# B&R Automation Studio project NAINV104C00R8L515F00 (part 24)

#### Act_Main.st - Do Not Change!!!
```iecst
(** 2020-05-26 **)
ACTION Act_Main:

	//Main
IF bModuleNotOK = FALSE THEN

		CASE eStat OF

			AWActIdle:
				IF eStatus <> Idle THEN	//Reset Data
					//Private
					fbStop(bEn := FALSE);
					fbRstAxisErr(bEn := FALSE);
					fbJog(bEn := FALSE);
					fbMovRel(bEn := FALSE);
					fbMovAbs(bEn := FALSE);
					fbHoming(bEn := FALSE);
					fbPwrOff(bEn := FALSE);
					fbPwrOn(bEn := FALSE);
					fbFullHm(bEn := FALSE);
					fbFullMovAbs(bEn := FALSE);
					fbFullMovAbsBl(bEn := FALSE);
					fbSDOWrite(bEn := FALSE);
					fbTm(IN := FALSE);
					usiStep				:= 0;
					usiCount			:= 0;
					bNotInterruptible	:= FALSE;
					tyParamOutDriver.uiCtrlword_6040.7	:= FALSE;
					sStatTxt	:= a_sStatText[eStat];

				END_IF

				eStatus	:= Idle;

				IF EDGENEG(p_bManual) THEN
					fMotionCANRstCtrlWord(ADR(tyParamOutDriver));
				END_IF

			AWActGoWidth:
				IF (eStatus = Idle OR eStatus = Busy) THEN

					eStatus	:= Busy;

					sStatTxt	:= a_sStatText[eStat];

					bNotInterruptible	:= TRUE;

					CASE usiStep OF
						0:	//Wait For Motion Parameter Update
							p_diMovePosInUM	:= fAWWidthToPosInUM(p_diGoWidth , p_diWidthAtHmPos);
							usiStep	:= 1;

						1:	//Check Position Difference
							IF tyParamOut.bPosDiff = TRUE THEN
								usiStep	:= 2;
							ELSE
								eStatus	:= Done;
							END_IF

						2:	//Move
							fbFullMovAbsBl.tyParamInDriver					:= tyParamInDriver;
							fbFullMovAbsBl.tyParamInMove.diPosInUM			:= p_diMovePosInUM;
							fbFullMovAbsBl.tyParamInMove.diDistInUM			:= p_diMoveDistInUM;
							fbFullMovAbsBl.tyParamInMove.diVelInUMPS		:= p_diMoveVelInUMPS;
							fbFullMovAbsBl.tyParamInMove.diAcc				:= p_diMoveAcc;
							fbFullMovAbsBl.tyParamInMove.diDec				:= p_diMoveDec;
							fbFullMovAbsBl.tyParamOut						:= tyParamOut;
							fbFullMovAbsBl(bEn := TRUE);

							IF fbFullMovAbsBl.udiStatus = 0 THEN
								eStatus	:= Done;
							ELSIF fbFullMovAbsBl.udiStatus < 65534 THEN
								eStatus		:= Error;

								IF fbFullMovAbsBl.udiStatus = 1401 THEN
									udiStatus	:= 10002;	//Power On Time Out While Going New Width
								ELSIF fbFullMovAbsBl.udiStatus = 1402 THEN
									udiStatus	:= 10003;	//Homing Time Out While Going New Width
								ELSIF fbFullMovAbsBl.udiStatus = 1403 THEN
									udiStatus	:= 10004;	//Move Absolute Time Out While Going New Width
								ELSIF fbFullMovAbsBl.udiStatus = 1405 THEN
									udiStatus	:= 10005;	//Stop Motion Time Out While Going New Width
								ELSIF fbFullMovAbsBl.udiStatus = 1408 THEN
									udiStatus	:= 10006;	//Axis Error Reset Failed While Going New Width
								ELSIF fbFullMovAbsBl.udiStatus = 1409 THEN
									udiStatus	:= 10007;	//Axis Error Occur In Move Absolute While Going New Width
								ELSIF fbFullMovAbsBl.udiStatus = 1411 THEN
									udiStatus	:= 10008;	//Axis Error Occur In Homing While Going New Width
								ELSIF fbFullMovAbsBl.udiStatus = 1412 THEN
									udiStatus	:= 10009;	//Homing Done But Home Flag Is Not Activated While Going New Width
								ELSIF fbFullMovAbsBl.udiStatus = 1413 THEN
									udiStatus	:= 10010;	//Forward Limit Activated In Homing While Going New Width
								ELSIF fbFullMovAbsBl.udiStatus = 1414 THEN
									udiStatus	:= 10011;	//Reverse Limit Activated In Homing While Going New Width
								ELSIF fbFullMovAbsBl.udiStatus = 1415 THEN
									udiStatus	:= 10012;	//Forward Limit Activated In Move Absolute While Going New Width
								ELSIF fbFullMovAbsBl.udiStatus = 1416 THEN
									udiStatus	:= 10013;	//Reverse Limit Activated In Move Absolute While Going New Width
								ELSE
									udiStatus	:= fbFullMovAbsBl.udiStatus;
								END_IF
							END_IF

					END_CASE

				END_IF

			AWActGoWidthOff:
				IF (eStatus = Idle OR eStatus = Busy) THEN

					eStatus	:= Busy;

					sStatTxt	:= a_sStatText[eStat];

					bNotInterruptible	:= TRUE;

					CASE usiStep OF
						0:	//Wait For Motion Parameter Update
							p_diMovePosInUM	:= fAWWidthToPosInUM(p_diGoWidth , p_diWidthAtHmPos);
							usiStep	:= 1;

						1:	//Check Position Difference
							IF tyParamOut.bPosDiff = TRUE THEN
								usiStep	:= 2;
							ELSE
								eStatus	:= Done;
							END_IF

						2:	//Move
							fbFullMovAbsBl.tyParamInDriver					:= tyParamInDriver;
							fbFullMovAbsBl.tyParamInMove.diPosInUM			:= p_diMovePosInUM;
							fbFullMovAbsBl.tyParamInMove.diDistInUM			:= p_diMoveDistInUM;
							fbFullMovAbsBl.tyParamInMove.diVelInUMPS		:= p_diMoveVelInUMPS;
							fbFullMovAbsBl.tyParamInMove.diAcc				:= p_diMoveAcc;
							fbFullMovAbsBl.tyParamInMove.diDec				:= p_diMoveDec;
							fbFullMovAbsBl.tyParamOut						:= tyParamOut;
							fbFullMovAbsBl(bEn := TRUE);

							IF fbFullMovAbsBl.udiStatus = 0 THEN
								usiStep	:= 3;
							ELSIF fbFullMovAbsBl.udiStatus < 65534 THEN
								eStatus		:= Error;

								IF fbFullMovAbsBl.udiStatus = 1401 THEN
									udiStatus	:= 10035;	//Power On Time Out While Going New Width And Off
								ELSIF fbFullMovAbsBl.udiStatus = 1402 THEN
									udiStatus	:= 10036;	//Homing Time Out While Going New Width And Off
								ELSIF fbFullMovAbsBl.udiStatus = 1403 THEN
									udiStatus	:= 10037;	//Move Absolute Time Out While Going New Width And Off
								ELSIF fbFullMovAbsBl.udiStatus = 1405 THEN
									udiStatus	:= 10038;	//Stop Motion Time Out While Going New Width And Off
								ELSIF fbFullMovAbsBl.udiStatus = 1408 THEN
									udiStatus	:= 10039;	//Axis Error Reset Failed While Going New Width And Off
								ELSIF fbFullMovAbsBl.udiStatus = 1409 THEN
									udiStatus	:= 10040;	//Axis Error Occur In Move Absolute While Going New Width And Off
								ELSIF fbFullMovAbsBl.udiStatus = 1411 THEN
									udiStatus	:= 10041;	//Axis Error Occur In Homing While Going New Width And Off
								ELSIF fbFullMovAbsBl.udiStatus = 1412 THEN
									udiStatus	:= 10042;	//Homing Done But Home Flag Is Not Activated While Going New Width And Off
								ELSIF fbFullMovAbsBl.udiStatus = 1413 THEN
									udiStatus	:= 10043;	//Forward Limit Activated In Homing While Going New Width And Off
								ELSIF fbFullMovAbsBl.udiStatus = 1414 THEN
									udiStatus	:= 10044;	//Reverse Limit Activated In Homing While Going New Width And Off
								ELSIF fbFullMovAbsBl.udiStatus = 1415 THEN
									udiStatus	:= 10045;	//Forward Limit Activated In Move Absolute While Going New Width And Off
								ELSIF fbFullMovAbsBl.udiStatus = 1416 THEN
									udiStatus	:= 10046;	//Reverse Limit Activated In Move Absolute While Going New Width And Off
								ELSE
									udiStatus	:= fbFullMovAbsBl.udiStatus;
								END_IF
							END_IF

						3:	//Turn Off Motor
							fMotionCANRstCtrlWord(ADR(tyParamOutDriver));
							eStatus	:= Done;

					END_CASE

				END_IF

			AWActFullHm:
				IF (eStatus = Idle OR eStatus = Busy) THEN

					eStatus	:= Busy;

					sStatTxt	:= a_sStatText[eStat];

					bNotInterruptible	:= TRUE;

					fbFullHm.tyParamInDriver	:= tyParamInDriver;
					fbFullHm.tyParamOut			:= tyParamOut;
					fbFullHm(bEn := TRUE);

					IF fbFullHm.udiStatus = 0 THEN
						eStatus	:= Done;
					ELSIF fbFullHm.udiStatus < 65534 THEN
						eStatus		:= Error;

						IF fbFullHm.udiStatus = 1401 THEN
							udiStatus	:= 10014;	//Power On Time Out While Full Homing
						ELSIF fbFullHm.udiStatus = 1402 THEN
							udiStatus	:= 10015;	//Homing Time Out While Full Homing
						ELSIF fbFullHm.udiStatus = 1405 THEN
							udiStatus	:= 10016;	//Stop Motion Time Out While Full Homing
						ELSIF fbFullHm.udiStatus = 1408 THEN
							udiStatus	:= 10017;	//Axis Error Reset Failed While Full Homing
						ELSIF fbFullHm.udiStatus = 1411 THEN
							udiStatus	:= 10018;	//Axis Error Occur In Homing While Full Homing
						ELSIF fbFullHm.udiStatus = 1412 THEN
							udiStatus	:= 10019;	//Homing Done But Home Flag Is Not Activated While Full Homing
						ELSIF fbFullHm.udiStatus = 1413 THEN
							udiStatus	:= 10020;	//Forward Limit Activated In Homing While Full Homing
						ELSIF fbFullHm.udiStatus = 1414 THEN
							udiStatus	:= 10021;	//Reverse Limit Activated In Homing While Full Homing
						ELSE
							udiStatus	:= fbFullHm.udiStatus;
						END_IF
					END_IF

				END_IF

			AWActPwrOn:
				IF (eStatus = Idle OR eStatus = Busy) THEN

					eStatus	:= Busy;

					sStatTxt	:= a_sStatText[eStat];

					fbPwrOn.tyParamInDriver	:= tyParamInDriver;
					fbPwrOn(bEn := TRUE);

					IF fbPwrOn.udiStatus = 0 THEN
						eStatus	:= Done;
					ELSIF fbPwrOn.udiStatus < 65534 THEN
						eStatus		:= Error;

						IF fbPwrOn.udiStatus = 1401 THEN
							udiStatus	:= 10022;	//Power On Time Out
						ELSE
							udiStatus	:= fbPwrOn.udiStatus;
						END_IF
					END_IF

				END_IF

			AWActPwrOff:
				IF (eStatus = Idle OR eStatus = Busy) THEN

					eStatus	:= Busy;

					sStatTxt	:= a_sStatText[eStat];

					fbPwrOff.tyParamInDriver	:= tyParamInDriver;
					fbPwrOff(bEn := TRUE);

					IF fbPwrOff.udiStatus = 0 THEN
						eStatus	:= Done;
					ELSIF fbPwrOff.udiStatus < 65534 THEN
						eStatus		:= Error;

						IF fbPwrOff.udiStatus = 1400 THEN
							udiStatus	:= 10023;	//Power Off Time Out
						ELSE
							udiStatus	:= fbPwrOff.udiStatus;
						END_IF
					END_IF

				END_IF

			AWActHoming:

				IF (eStatus = Idle OR eStatus = Busy) THEN

					eStatus	:= Busy;

					sStatTxt	:= a_sStatText[eStat];

					bNotInterruptible	:= TRUE;

					fbHoming.tyParamInDriver	:= tyParamInDriver;
					fbHoming.tyParamOut			:= tyParamOut;
					fbHoming(bEn := TRUE);

					IF fbHoming.udiStatus = 0 THEN
						eStatus	:= Done;
					ELSIF fbHoming.udiStatus < 65534 THEN
						eStatus		:= Error;

						IF fbHoming.udiStatus = 1402 THEN
							udiStatus	:= 10024;	//Homing Time Out
						ELSIF fbHoming.udiStatus = 1411 THEN
							udiStatus	:= 10018;	//Axis Error Occur In Homing While Full Homing

						ELSIF fbHoming.udiStatus = 1413 THEN
							udiStatus	:= 10020;	//Forward Limit Activated In Homing While Full Homing
						ELSIF fbHoming.udiStatus = 1414 THEN
							udiStatus	:= 10021;	//Reverse Limit Activated In Homing While Full Homing
						ELSE
							udiStatus	:= fbHoming.udiStatus;
						END_IF
					END_IF

				END_IF

			AWActMovAbs:
				IF (eStatus = Idle OR eStatus = Busy) THEN

					eStatus	:= Busy;

					sStatTxt	:= a_sStatText[eStat];

					bNotInterruptible	:= TRUE;

					fbMovAbs.tyParamInDriver			:= tyParamInDriver;
					fbMovAbs.tyParamInMove.diPosInUM	:= p_diMovePosInUM;
					fbMovAbs.tyParamInMove.diDistInUM	:= p_diMoveDistInUM;
					fbMovAbs.tyParamInMove.diVelInUMPS	:= p_diMoveVelInUMPS;
					fbMovAbs.tyParamInMove.diAcc		:= p_diMoveAcc;
					fbMovAbs.tyParamInMove.diDec		:= p_diMoveDec;
					fbMovAbs(bEn := TRUE);

					IF fbMovAbs.udiStatus = 0 THEN
						eStatus	:= Done;
					ELSIF fbMovAbs.udiStatus < 65534 THEN
						eStatus		:= Error;

						IF fbMovAbs.udiStatus = 1403 THEN
							udiStatus	:= 10025;	//Move Absolute Time Out
						ELSE
							udiStatus	:= fbMovAbs.udiStatus;
						END_IF
					END_IF

				END_IF

			AWActMovRel:
				IF (eStatus = Idle OR eStatus = Busy) THEN

					eStatus	:= Busy;

					sStatTxt	:= a_sStatText[eStat];

					bNotInterruptible	:= TRUE;

					fbMovRel.tyParamInDriver			:= tyParamInDriver;
					fbMovRel.tyParamInMove.diPosInUM	:= p_diMovePosInUM;
					fbMovRel.tyParamInMove.diDistInUM	:= p_diMoveDistInUM;
					fbMovRel.tyParamInMove.diVelInUMPS	:= p_diMoveVelInUMPS;
					fbMovRel.tyParamInMove.diAcc		:= p_diMoveAcc;
					fbMovRel.tyParamInMove.diDec		:= p_diMoveDec;
					fbMovRel(bEn := TRUE);

					IF fbMovRel.udiStatus = 0 THEN
						eStatus	:= Done;
					ELSIF fbMovRel.udiStatus < 65534 THEN
						eStatus		:= Error;

						IF fbMovRel.udiStatus = 1404 THEN
							udiStatus	:= 10026;	//Move Relative Time Out
						ELSE
							udiStatus	:= fbMovRel.udiStatus;
						END_IF
					END_IF

				END_IF

			AWActJogOpen:
				IF (eStatus = Idle OR eStatus = Busy) THEN

					eStatus	:= Busy;

					sStatTxt	:= a_sStatText[eStat];

					bNotInterruptible	:= TRUE;

					fbJog.tyParamInDriver	:= tyParamInDriver;
					fbJog.tyParamInMove.diAcc		:= p_diMoveAcc;
					fbJog.tyParamInMove.diDec		:= p_diMoveDec;

					IF p_bDir = TRUE THEN
						fbJog.tyParamInJog.diVelInUMPS	:= p_diJogVelInUMPS;
					ELSE
						fbJog.tyParamInJog.diVelInUMPS	:= p_diJogVelInUMPS * -1;
					END_IF

					fbJog(bEn := TRUE);

					IF fbJog.udiStatus = 0 THEN
						bJogging	:= TRUE;
						bJogOpen	:= TRUE;
						eStatus		:= Done;
					ELSIF fbJog.udiStatus < 65534 THEN
						udiStatus	:= fbJog.udiStatus;
						eStatus		:= Error;
					END_IF

				END_IF

			AWActJogClose:
				IF (eStatus = Idle OR eStatus = Busy) THEN

					eStatus	:= Busy;

					sStatTxt	:= a_sStatText[eStat];

					bNotInterruptible	:= TRUE;

					fbJog.tyParamInDriver			:= tyParamInDriver;
					fbJog.tyParamInMove.diAcc		:= p_diMoveAcc;
					fbJog.tyParamInMove.diDec		:= p_diMoveDec;

					IF p_bDir = TRUE THEN
						fbJog.tyParamInJog.diVelInUMPS	:= p_diJogVelInUMPS * -1;
					ELSE
						fbJog.tyParamInJog.diVelInUMPS	:= p_diJogVelInUMPS;
					END_IF

					fbJog(bEn := TRUE);

					IF fbJog.udiStatus = 0 THEN
						bJogging	:= TRUE;
						bJogClose	:= TRUE;
						eStatus		:= Done;
					ELSIF fbJog.udiStatus < 65534 THEN
						udiStatus	:= fbJog.udiStatus;
						eStatus		:= Error;
					END_IF

				END_IF

			AWActJogStop:
				IF (eStatus = Idle OR eStatus = Busy) THEN

					sStatTxt	:= a_sStatText[eStat];

					fMotionCANJogStop(ADR(tyParamOutDriver));
					bJogging	:= FALSE;
					bJogClose	:= FALSE;
					bJogOpen	:= FALSE;
					eStatus	:= Done;

				END_IF

			AWActRstAxisErr:
				IF (eStatus = Idle OR eStatus = Busy) THEN

					eStatus	:= Busy;

					sStatTxt	:= a_sStatText[eStat];

					fbRstAxisErr(bEn := TRUE);

					IF fbRstAxisErr.udiStatus = 0 THEN
						eStatus	:= Done;
					ELSIF fbRstAxisErr.udiStatus < 65534 THEN
						udiStatus	:= fbRstAxisErr.udiStatus;
						eStatus		:= Error;
					END_IF

				END_IF

			AWActStop:
				IF (eStatus = Idle OR eStatus = Busy) THEN

					eStatus	:= Busy;

					sStatTxt	:= a_sStatText[eStat];

					fbStop.tyParamInDriver	:= tyParamInDriver;
					fbStop(bEn := TRUE);

					IF fbStop.udiStatus = 0 THEN
						bJogging	:= FALSE;
						bJogClose	:= FALSE;
						bJogOpen	:= FALSE;
						eStatus		:= Done;
					ELSIF fbStop.udiStatus < 65534 THEN
						eStatus		:= Error;

						IF fbStop.udiStatus = 1405 THEN
							udiStatus	:= 10027;	//Stop Motion Time Out
						ELSE
							udiStatus	:= fbStop.udiStatus;
						END_IF
					END_IF

				END_IF
		END_CASE

ELSE
	CASE eStat OF
		AWActSDOWrite:
			IF (eStatus = Idle OR eStatus = Busy) THEN

				eStatus	:= Busy;

				sStatTxt	:= a_sStatText[eStat];

				fbTm(IN := TRUE);

				IF fbTm.Q THEN

					fbSDOWrite.tyParamOut	:= tyParamOut;
					fbSDOWrite.tyTuning		:= p_tyTuning;

					fbSDOWrite(bEn := TRUE);

					IF fbSDOWrite.udiStatus = 0 THEN
						eStatus	:= Done;
					ELSIF fbSDOWrite.udiStatus < 65534 THEN
						fMotionCANRstCtrlWord(ADR(tyParamOutDriver));

						IF usiCount < 5 THEN
							fbTm(IN := FALSE);
							fbSDOWrite(bEn := FALSE);

							usiCount	:= usiCount + 1;
						ELSE
							eStatus	:= Error;

							IF fbSDOWrite.udiStatus = 1406 THEN
								udiStatus	:= 10028;	//SDO Write Error
							ELSE
								udiStatus	:= fbSDOWrite.udiStatus;
							END_IF
						END_IF

					END_IF

				END_IF

			END_IF

		AWActBGStartModOKChk:
			IF (eStatus = Idle OR eStatus = Busy) THEN

				sStatTxt	:= a_sStatText[eStat];

				bModuleOKChk	:= TRUE;
				eStatus			:= Done;

			END_IF

		AWActBGStopModOKChk:
			IF (eStatus = Idle OR eStatus = Busy) THEN

				sStatTxt	:= a_sStatText[eStat];

				bModuleOKChk	:= FALSE;
				eStatus			:= Done;

			END_IF

		AWActIdle:
			IF eStatus <> Idle THEN	//Reset Data
				//Private
				fbStop(bEn := FALSE);
				fbRstAxisErr(bEn := FALSE);
				fbJog(bEn := FALSE);
				fbMovRel(bEn := FALSE);
				fbMovAbs(bEn := FALSE);
				fbHoming(bEn := FALSE);
				fbPwrOff(bEn := FALSE);
				fbPwrOn(bEn := FALSE);
				fbFullHm(bEn := FALSE);
				fbFullMovAbs(bEn := FALSE);
				fbFullMovAbsBl(bEn := FALSE);
				fbSDOWrite(bEn := FALSE);
				fbTm(IN := FALSE);
				usiStep				:= 0;
				usiCount			:= 0;
				bNotInterruptible	:= FALSE;
				tyParamOutDriver.uiCtrlword_6040.7	:= FALSE;

				sStatTxt	:= a_sStatText[eStat];

			END_IF

			eStatus	:= Idle;

			IF EDGENEG(p_bManual) THEN
				fMotionCANRstCtrlWord(ADR(tyParamOutDriver));
			END_IF

		AWActRstNode:
			IF (eStatus = Idle OR eStatus = Busy) THEN

				eStatus	:= Busy;

				sStatTxt	:= a_sStatText[eStat];
				IF bRstErr THEN
					fbModuleOK(bEn := FALSE, bModuleOK := bModuleOK);
				END_IF
				fbModuleOK(bEn := TRUE);
				IF fbModuleOK.udiStatus = 0 THEN
					fbModuleOK(bEn := FALSE);
					eStatus			:= Done;
				ELSIF fbModuleOK.udiStatus < 65534 THEN
					eStatus		:= Error;

					IF fbModuleOK.udiStatus = 1407 THEN
						udiStatus	:= 10001;	//CANOpen Communication Error, ModuleOK Not TRUE
						fbModuleOK(bEn := FALSE);
					ELSE
						udiStatus	:= fbModuleOK.udiStatus;
					END_IF
				END_IF
			END_IF

		AWActRstAxisErr:
			IF (eStatus = Idle OR eStatus = Busy) THEN

				eStatus	:= Busy;

				sStatTxt	:= a_sStatText[eStat];

				fbRstAxisErr(bEn := TRUE);

				IF fbRstAxisErr.udiStatus = 0 THEN
					eStatus	:= Done;
				ELSIF fbRstAxisErr.udiStatus < 65534 THEN
					udiStatus	:= fbRstAxisErr.udiStatus;
					eStatus		:= Error;
				END_IF

			END_IF

	END_CASE
END_IF

END_ACTION
```

#### Act_Main_Disable.st - Do Not Change!!!
```iecst
(** 2020-03-16 **)
ACTION Act_Main_Disable:

	tyParamOut.bAxisErr			:= FALSE;
	tyParamOut.bFwdLmtSen		:= FALSE;
	tyParamOut.bInPos			:= TRUE;
	tyParamOut.bIsHomed			:= TRUE;
	tyParamOut.bPosDiff			:= FALSE;
	tyParamOut.bPwrOn			:= TRUE;
	tyParamOut.bRevLmtSen		:= FALSE;
	tyParamOut.bStopped			:= TRUE;
	tyParamOut.diActualPosInUM	:= 0;
	tyParamOut.diHmAcc			:= 0;
	tyParamOut.diHmSpdForSwitch	:= 0;
	tyParamOut.diHmSpdForZero	:= 0;
	tyParamOut.diProfileAcc		:= 0;
	tyParamOut.diProfileDec		:= 0;
	tyParamOut.udiAxisErrID		:= 0;

	bWidthPosDiff				:= FALSE;
	bModuleNotOK				:= FALSE;
END_ACTION
```

#### Act_Background.st - Do Not Change!!!
```iecst
(** 2020-05-26 **)
ACTION Act_Background:

	//Update Parameter
	IF bModuleOK = TRUE THEN

		tyParamInMove.diPosInUM		:= p_diMovePosInUM;
		tyParamInMove.diDistInUM	:= p_diMoveDistInUM;
		tyParamInMove.diVelInUMPS	:= p_diMoveVelInUMPS;
		tyParamInMove.diAcc			:= p_diMoveAcc;
		tyParamInMove.diDec			:= p_diMoveDec;

		fMotionCANUpdtDat(ADR(tyParamOut) , p_tyParamInConvert , tyParamOutDriver , tyParamInDriver , tyParamInMove , p_tyParamInHm , p_bDir, p_eNtParamMotorType);

		bWidthPosDiff	:= (tyParamOut.bIsHomed = FALSE) OR ((ABS((fAWWidthToPosInUM(p_diGoWidth , p_diWidthAtHmPos)) - tyParamOut.diActualPosInUM)) > 500);

		p_tyParamInConvert.diPitchInUM	:= fPitchCalc(p_diWidthOffsetInUM , p_diMaxWidthInUM , p_diMinWidthInUM , p_diPitchInUM);

		fbFullMovAbsBl.tyParamInConvert					:= p_tyParamInConvert;

		IF p_bDir = TRUE THEN
			bOpenSen	:= tyParamOut.bFwdLmtSen;
			bCloseSen	:= tyParamOut.bRevLmtSen;
		ELSE
			bOpenSen	:= tyParamOut.bRevLmtSen;
			bCloseSen	:= tyParamOut.bFwdLmtSen;
		END_IF

		CASE p_eNtParamMotorType OF
			DeltaAsdaA2:
				CASE tyParamOut.udiAxisErrID OF
					8976:	sAxisErrTxt	:= 'Over Current';
					12560:	sAxisErrTxt	:= 'Over Voltage';
					12576:	sAxisErrTxt	:= 'Under Voltage';
					12592:	sAxisErrTxt	:= 'Input Power Phase Loss';
					12816:	sAxisErrTxt	:= 'Regeneration Error';
					12848:	sAxisErrTxt	:= 'Overload';
					12849:	sAxisErrTxt	:= 'Pre-overload Warning';
					13056:	sAxisErrTxt	:= 'U,V,W Wiring Error';
					16912:	sAxisErrTxt	:= 'IGBT Temperature Error';
					21296:	sAxisErrTxt	:= 'Memory Error';
					21569:	sAxisErrTxt	:= 'Emergency Stop Activated';
					21570:	sAxisErrTxt	:= 'Forward Limit Switch Error';
					21571:	sAxisErrTxt	:= 'Reverse Limit Switch Error';
					21572:	sAxisErrTxt	:= 'Forward Software Limit';
					21573:	sAxisErrTxt	:= 'Reverse Software Limit';
					21760:	sAxisErrTxt	:= 'DSP Firmware Upgrade';
					25088:	sAxisErrTxt	:= 'CANopen SYNC Error';
					25360:	sAxisErrTxt	:= 'CANopen Data Initial Error';
					25376:	sAxisErrTxt	:= 'Adjustment Error';
					28961:	sAxisErrTxt	:= 'Motor Protection Error';
					28962:	sAxisErrTxt	:= 'Motor Error';
					29445:	sAxisErrTxt	:= 'Encoder Error';
					29446:	sAxisErrTxt	:= 'Encoder Output Error';
					29968:	sAxisErrTxt	:= 'Serial Communication Error';
					29984:	sAxisErrTxt	:= 'Serial Communication Time Out';
					33024:	sAxisErrTxt	:= 'CANbus Error (Bus-off)';
					33040:	sAxisErrTxt	:= 'CANopen SDO receive buffer overrun';
					33056:	sAxisErrTxt	:= 'CANbus Error (Warning)';
					33072:	sAxisErrTxt	:= 'Node Guarding or Heartbeat Error';
					33280:	sAxisErrTxt	:= 'CANopen PDO Object Error';
					33792:	sAxisErrTxt	:= 'Over Speed';
					34304:	sAxisErrTxt	:= 'Abnormal Pulse Control Command';
					34320:	sAxisErrTxt	:= 'Full Closed Loop Excessive Deviation';
					34321:	sAxisErrTxt	:= 'Excessive Deviation';
				END_CASE

			SchneiderLexium28:
				CASE tyParamOut.udiAxisErrID OF
					8724:	sAxisErrTxt	:= 'Over Current';
					8976:	sAxisErrTxt	:= 'Motor Overload';
					8977:	sAxisErrTxt	:= 'Drive overload (foldback)';
					9088:	sAxisErrTxt	:= 'Calculated offsets for current sensors out OF range';
					9089:	sAxisErrTxt := 'Motor phase missing';
					9090:	sAxisErrTxt := 'Overcurrent detected at one OF the digital outputs';
					12560:	sAxisErrTxt	:= 'DC Bus Over Voltage';
					12576:	sAxisErrTxt	:= 'DC Bus Under Voltage';
					12672:	sAxisErrTxt	:= 'Braking Resistor Overload';
					12673:	sAxisErrTxt	:= 'Safety function Safe Torque Off (STO) triggered';
					12674:	sAxisErrTxt	:= 'DC bus voltage measurement';
					12675:	sAxisErrTxt	:= 'Missing mains supply, undervoltage mains supply';
					12676:	sAxisErrTxt := 'The encoder supply voltage has dropped under operational value';
					12677:	sAxisErrTxt := 'The multi turn encoder battery voltage has dropped under 3 Vdc';
					12678:	sAxisErrTxt := 'Internal position synchronization error	detected between the multi turn AND the single turn modules';
					12679:	sAxisErrTxt := 'Generic error code of the multi turn module is detected';
					12697:	sAxisErrTxt := 'Braking resistor overload';
					16512:	sAxisErrTxt	:= 'Drive overtemperature (IPM)';
					16513:	sAxisErrTxt	:= 'Drive overtemperature (controller)';
					16534:	sAxisErrTxt := 'Temperature sensor inoperative';
					17168:	sAxisErrTxt	:= 'Power stage overtemperature';
					17280:	sAxisErrTxt := 'The encoder temperature is too high';
					17424:	sAxisErrTxt	:= 'Motor overtemperature';
					21808:	sAxisErrTxt	:= 'System error detected (nonvolatilememory)';
					21893:	sAxisErrTxt	:= 'Error detected in non-volatile memory';
					21889:	sAxisErrTxt	:= 'System error detected (nonvolatile memory)';
					21890:	sAxisErrTxt	:= 'System error detected (CAN power supply)';
					21891:	sAxisErrTxt	:= 'System error detected (selftest)';
					21894:	sAxisErrTxt	:= 'System error detected (NV ACCESS)';
					25472:	sAxisErrTxt	:= 'Target position rejected';
					25985:	sAxisErrTxt	:= 'System error detected(FPGA)';
					28816:	sAxisErrTxt	:= 'System error detected (FPGA does NOT match firmware)';
					28817:	sAxisErrTxt	:= 'Emergency Stop Activated';
					28961:	sAxisErrTxt := 'Motor blocked';
					29080:	sAxisErrTxt := 'Commutation error detected';
					29568:  sAxisErrTxt	:= 'Error detected in communication with motor encoder';
					29574:	sAxisErrTxt	:= 'Drive is not synchronous wit master cycle';
					29581:	sAxisErrTxt := 'System error detected (encoder)';
					29587:	sAxisErrTxt	:= 'Encoder overvoltage or overcurrent';
					29592:	sAxisErrTxt := 'The returned position value are no longer considered valid';
					29593:	sAxisErrTxt := 'The multi turn encoder requires an explicit configuration command';
					30081:	sAxisErrTxt := 'Target position rejected';
					30082:	sAxisErrTxt := 'No target values received via the fieldbus';
					33072:	sAxisErrTxt	:= 'CANopen: Heartbeat error detected';
					33296:	sAxisErrTxt := 'R_PDO is too short';
					33921:	sAxisErrTxt	:= 'Actual Motor Velocity Too High';
					33553:	sAxisErrTxt	:= 'Motor torque too high FOR an excessive period OF time';
					33664:	sAxisErrTxt := 'Unstable current loop';
					33922:	sAxisErrTxt := 'Velocity deviation too high';
					34321:	sAxisErrTxt	:= 'Position deviation too high';
					34432:	sAxisErrTxt := 'Position deviation via signal output function MC_OK';
					34441:	sAxisErrTxt := 'Position deviation too high (following error)';
					61568:	sAxisErrTxt	:= 'Fieldbus: Communication	error detected';
					65282:	sAxisErrTxt	:= 'Not possible to read data of electronic motor nameplate';
					65296:	sAxisErrTxt	:= 'Forward Limit Switch Error';
					65297:	sAxisErrTxt	:= 'Reverse Limit Switch Error';
					65281:	sAxisErrTxt := 'System error detected';
					65298:	sAxisErrTxt	:= 'Forward Software Limit';
					65299:	sAxisErrTxt	:= 'Reverse Software Limit';
					65301:	sAxisErrTxt := 'The encoder firmware cannot operate on the provided hardware';

				END_CASE

			EstunPronet:
				CASE tyParamOut.udiAxisErrID OF
					65281:	sAxisErrTxt	:= 'Parameter breakdown';//A01
					65282:	sAxisErrTxt	:= 'AD shift channels breakdown';
					65283:	sAxisErrTxt	:= 'Overspeed';
					65284:	sAxisErrTxt	:= 'Overload';
					65285:	sAxisErrTxt := 'Position error counteroverflow ';
					65286:	sAxisErrTxt := 'Position error pulse overflow';
					65287:	sAxisErrTxt	:= 'The setting of electronic gear or given pulse frequency is not reasonable';
					65288:	sAxisErrTxt	:= 'The 1st channel of current detection is wrong.';
					65289:	sAxisErrTxt	:= 'The 2nd channel of current detection is wrong.';
					65290:	sAxisErrTxt	:= 'Incremental Encoder is break off.';//A10
					65292:	sAxisErrTxt	:= 'Overcurrent';
					65293:	sAxisErrTxt	:= 'Overvoltage';
					65294:	sAxisErrTxt	:= 'Undervoltage';
					65295:	sAxisErrTxt := 'Bleeder resistor error';
					65296:	sAxisErrTxt := 'Regeneration error';
					65297:	sAxisErrTxt := 'Resolver error';
					65298:	sAxisErrTxt := 'IGBT superheat alarm';
					65299:	sAxisErrTxt := 'Motor overheat alarm';
					65300:	sAxisErrTxt := 'Power line phase shortage';//A20
					65301:	sAxisErrTxt	:= 'Instantaneous power off alarm';
					65302:	sAxisErrTxt	:= 'Motor temperature detection sensor is break off.';
					65303:	sAxisErrTxt := 'Brake overcurrent alarm';//A23
					65305:	sAxisErrTxt := 'Motor power line U overcurrent';//A25
					65306:	sAxisErrTxt := 'Motor power line V overcurrent';//A26
					65307:	sAxisErrTxt := 'Motor power line W overcurrent';//A27
					65322:	sAxisErrTxt	:= 'Servomotor type error';//A42
					65323:	sAxisErrTxt	:= 'Servo drive type error';
					65325:	sAxisErrTxt	:= 'Absolute encoder multiturn information error';
					65326:	sAxisErrTxt	:= 'Absolute encoder multiturn information overflow';
					65327:	sAxisErrTxt	:= 'Battery voltage below 2.5V';
					65328:	sAxisErrTxt	:= 'Battery voltage below 3.1V';//A48
					65330:	sAxisErrTxt := 'Serial encoder communication overtime ';//A50
					65331:	sAxisErrTxt := 'Absolute encoder overspeed alarm detected';
					65332:  sAxisErrTxt	:= 'Absolute state of serial encoder error';
					65333:	sAxisErrTxt	:= 'Serial encoder calcaution error';
					65334:	sAxisErrTxt := 'Parity bit or end bit in serial encoder control domain error';
					65335:	sAxisErrTxt	:= 'Serial encoder communication data checking error';
					65336:	sAxisErrTxt := 'End bit in serial encoder control domain error';
					65338:	sAxisErrTxt := 'Serial encoder data empty';
					65339:	sAxisErrTxt := 'Serial encoder data format error';
					65340:	sAxisErrTxt := 'Communication module not detected ';//A60
					65341:	sAxisErrTxt := 'Communication unsuccessful';
					65342:	sAxisErrTxt := 'Servo drive can not receive the period data of communication module ';
					65343:	sAxisErrTxt := 'Communication module can not receive the servo drive response data.';
					65344:	sAxisErrTxt := 'Communication module and bus connectionless';
					65346:	sAxisErrTxt := 'CAN communication abnormal';
					65347:	sAxisErrTxt := 'Receiving heartbeat timeout';
					65349:	sAxisErrTxt := 'Synchronization signal monitoring cycle is longer than setting';
					65362: sAxisErrTxt := 'Torque output alarm';
				END_CASE
		END_CASE

	ELSE

		tyParamOut.bAxisErr			:= FALSE;
		tyParamOut.bFwdLmtSen		:= FALSE;
		tyParamOut.bInPos			:= FALSE;
		tyParamOut.bIsHomed			:= FALSE;
		tyParamOut.bPosDiff			:= TRUE;
		tyParamOut.bPwrOn			:= FALSE;
		tyParamOut.bRevLmtSen		:= FALSE;
		tyParamOut.bStopped			:= TRUE;
		tyParamOut.diActualPosInUM	:= 0;
		tyParamOut.diHmAcc			:= 0;
		tyParamOut.diHmSpdForSwitch	:= 0;
		tyParamOut.diHmSpdForZero	:= 0;
		tyParamOut.diProfileAcc		:= 0;
		tyParamOut.diProfileDec		:= 0;
		tyParamOut.udiAxisErrID		:= 0;

		bWidthPosDiff				:= TRUE;

	END_IF

	//Abnormal Movement
	IF eStatus1 <> Error THEN
		IF p_bOps = TRUE AND eStatus = Idle THEN
			IF (ABS(tyParamOut.diActualPosInUM - diActualPosInUMOld) > 2000) AND (ABS(tyParamOut.diActualPosInUM - diActualPosInUMOld) < 10000) THEN
				eStatus1	:= Error;
				udiStatus1	:= 10000;	//Axis Move Abnormally By External Force

				fMotionCANRstCtrlWord(ADR(tyParamOutDriver));
				p_eAct	:= AWActIdle;
				eStat	:= AWActIdle;
			END_IF
		ELSE
			diActualPosInUMOld	:= tyParamOut.diActualPosInUM;
		END_IF
	END_IF

	//Reset Error
	IF (eStatus1 = Error) AND bRstErr THEN
		eStatus1	:= Idle;
		udiStatus1	:= 0;
	END_IF

	//Request Position To Movement Out Of Range
	IF p_bOps
		AND((tyParamInMove.diPosInUM < p_diMinAbsPosInUM) OR (tyParamInMove.diPosInUM > p_diMaxAbsPosInUM))
		AND (eStatus2 <> Error) THEN
		eStatus2	:= Error;
		udiStatus2	:= 10029;	//Request Absolute Position Out Of Range

		fMotionCANRstCtrlWord(ADR(tyParamOutDriver));
		p_eAct	:= AWActIdle;
		eStat	:= AWActIdle;
	END_IF

	//Reset Error
	IF (eStatus2 = Error) AND bRstErr THEN
		eStatus2	:= Idle;
		udiStatus2	:= 0;
	END_IF

	//Sensor Interrupt
	IF bNotInterruptible = TRUE AND eStatus3 <> Error THEN

		IF p_bInletSensor = TRUE THEN
			eStatus3	:= Error;
			udiStatus3	:= 10030;	//Inlet Sensor Interrupt Auto Width Movement

			fMotionCANRstCtrlWord(ADR(tyParamOutDriver));
			p_eAct	:= AWActIdle;
			eStat	:= AWActIdle;

		ELSIF p_bOutletSensor = TRUE THEN
			eStatus3	:= Error;
			udiStatus3	:= 10031;	//Outlet Sensor Interrupt Auto Width Movement

			fMotionCANRstCtrlWord(ADR(tyParamOutDriver));
			p_eAct	:= AWActIdle;
			eStat	:= AWActIdle;

		ELSIF p_bClearSensor = TRUE THEN
			eStatus3	:= Error;
			udiStatus3	:= 10032;	//Clear Sensor Interrupt Auto Width Movement

			fMotionCANRstCtrlWord(ADR(tyParamOutDriver));
			p_eAct	:= AWActIdle;
			eStat	:= AWActIdle;

		ELSIF p_bMiddleSensor = TRUE THEN
			eStatus3	:= Error;
			udiStatus3	:= 10033;	//Middle Sensor Interrupt Auto Width Movement

			fMotionCANRstCtrlWord(ADR(tyParamOutDriver));
			p_eAct	:= AWActIdle;
			eStat	:= AWActIdle;

		ELSIF p_bInterruptSensor = TRUE THEN
			eStatus3	:= Error;
			udiStatus3	:= 10034;	//Sensor Interrupt Auto Width Movement

			fMotionCANRstCtrlWord(ADR(tyParamOutDriver));
			p_eAct	:= AWActIdle;
			eStat	:= AWActIdle;

		ELSIF p_bCloseInterruptSensor = TRUE AND bJogOpen = FALSE THEN
			eStatus3	:= Error;
			udiStatus3	:= 10047;	//Sensor Interrupt Auto Width Movement

			fMotionCANRstCtrlWord(ADR(tyParamOutDriver));
			p_eAct	:= AWActIdle;
			eStat	:= AWActIdle;

		ELSIF p_bOpenInterruptSensor = TRUE AND bJogClose = FALSE THEN
			eStatus3	:= Error;
			udiStatus3	:= 10048;	//Sensor Interrupt Auto Width Movement

			fMotionCANRstCtrlWord(ADR(tyParamOutDriver));
			p_eAct	:= AWActIdle;
			eStat	:= AWActIdle;
		END_IF

	END_IF

	//Reset Error
	IF (eStatus3 = Error AND bRstErr)
		OR (p_bOpenInterruptSensor AND eStat = AWActJogClose)
		OR (p_bCloseInterruptSensor AND eStat = AWActJogOpen)
		THEN
		eStatus3	:= Idle;
		udiStatus3	:= 0;
	END_IF

	IF bRstErr THEN
		udiStatus	:= 0;
		bJogging	:= FALSE;
		bJogClose	:= FALSE;
		bJogOpen	:= FALSE;
	END_IF

	fbServoModuleOk(IN:= bModuleOK);
	fbServoModuleNotOk(IN:= bModuleOK = FALSE);
	IF fbServoModuleNotOk.Q AND udiStatus <> 10001 THEN

		bModuleNotOK		:= TRUE;
		bModuleNotOKLock	:= TRUE;
		usiRstStep	:= 0;
		tyParamOutDriver.uiCtrlword_6040	:= 0;
		tyParamOutDriver.siModOfOpt_6060	:= 0;
		tyParamOutDriver.diTargetPos_607A	:= 0;
		tyParamOutDriver.udiMoveSpd_6081	:= 0;
		tyParamOutDriver.siHmMethod_6098	:= 0;
		tyParamOutDriver.diJogVel_60FF		:= 0;

		CASE p_eNtParamMotorType OF

			DeltaAsdaA2:
				fbModuleOK(bModuleOK:= FALSE);
				IF eStatus = Idle THEN
					eAct	:= AWActRstNode;
				END_IF

				IF (eStatus = Done OR eStatus = Error)AND eStat = AWActRstNode THEN

					eAct	:= AWActIdle;
				END_IF

			EstunPronet:
				fbModuleOK(bModuleOK:= FALSE);
				IF eStatus = Idle THEN
					eAct	:= AWActRstNode;
				END_IF

				IF (eStatus = Done OR eStatus = Error)AND eStat = AWActRstNode THEN

					eAct	:= AWActIdle;
				END_IF

			SchneiderLexium28:
			// Do Nothing
		END_CASE

	ELSIF bModuleNotOK = TRUE AND fbServoModuleOk.Q THEN

		CASE usiRstStep OF

			0:
				IF eStatus = Idle THEN
					eAct	:= AWActRstAxisErr;
				END_IF

				IF eStatus = Done AND eStat = AWActRstAxisErr THEN
					eAct	:= AWActIdle;
					usiRstStep	:= 4;
				END_IF

			4: tyParamOutDriver.siModOfOpt_6060 := 1;
				usiRstStep	:= 5;

			5: tyParamOutDriver.siModOfOpt_6060 := 1;
				fbRstNodeTimer(IN:=TRUE);

				IF tyParamInDriver.siModOfOptDisp_6061 = 1 THEN
					usiRstStep	:= 6;
					fbRstNodeTimer(IN:=FALSE);
				ELSIF fbRstNodeTimer.Q THEN
					usiRstStep	:= 8;
					fbRstNodeTimer(IN:=FALSE);
				END_IF

			6: tyParamOutDriver.siModOfOpt_6060 := 6;
				fbRstNodeTimer(IN:=FALSE);
				usiRstStep	:= 7;

			7: tyParamOutDriver.siModOfOpt_6060 := 6;
				fbRstNodeTimer(IN:=TRUE);

				IF tyParamInDriver.siModOfOptDisp_6061 = 6 THEN
					usiRstStep	:= 10;
					fbRstNodeTimer(IN:=FALSE);
				ELSIF fbRstNodeTimer.Q THEN
					usiRstStep	:= 9;
					fbRstNodeTimer(IN:=FALSE);
				END_IF

			8:	fbModuleOK(bEn := TRUE, bModuleOK:= FALSE);
				fbRstNodeTimer(IN:=FALSE);
				usiRstStep	:= 9;

			9:	fbModuleOK(bModuleOK:= FALSE);
				IF eStatus = Idle THEN
					eAct	:=AWActRstNode;
				END_IF

				IF eStatus = Done AND eStat = AWActRstNode THEN
					usiRstStep	:= 0;
					eAct		:= AWActIdle;
				END_IF

			10:IF eStatus = Idle THEN
					eAct	:= AWActRstAxisErr;
				END_IF

				IF eStatus = Done AND eStat = AWActRstAxisErr THEN
					eAct			:=AWActIdle;
					usiRstStep	:= 11;
				END_IF

			11:

				IF eStatus = Idle THEN
					eAct	:= AWActSDOWrite;
				END_IF

				IF eStatus = Done AND eStat = AWActSDOWrite THEN
					eAct			:= AWActIdle;
					usiRstStep	:= 13;

				ELSIF udiStatus = 10028 THEN
					eAct			:= AWActIdle;
					usiRstStep	:= 0;
				END_IF

			13: bModuleNotOK	:= FALSE;
				usiRstStep	:= 0;
		END_CASE
	ELSE
		eAct	:= AWActIdle;

	END_IF

	IF tyParamOut.bPosDiff = FALSE THEN
		tyParamOutDriver.uiCtrlword_6040.4	:= FALSE;
	END_IF

END_ACTION
```

#### Act_CombineErr.st - Do Not Change!!!
```iecst
(** 2020-03-16 **)
ACTION Act_CombineErr:

	//Combine Error
	IF eStatus = Error OR eStatus1 = Error OR eStatus2 = Error OR eStatus3 = Error THEN
		eMainStatus	:= Error;
	ELSE
		eMainStatus	:= eStatus;
	END_IF

END_ACTION
```

#### Act_Alarm.st - Do Not Change!!!
```iecst
(** 2020-03-16 **)
ACTION Act_Alarm:

	//Error
	IF EDGEPOS(eStatus = Error) THEN

		tyAlmData.sProgNm		:= p_sProgNm;
		tyAlmData.udiCode		:= udiStatus;
		tyAlmData.eSeverity		:= AlmSeverityError;
		tyAlmData.udiRunTime	:= tyAlmData.udiRunTime + 1;
		tyAlmData.bAlm			:= TRUE;
		tyAlmData.udiModuleNum  := udiModuleNum;
		g_sAWOpenProgNm:= p_sProgNm;

		//Get Error Message
		IF tyAlmData.udiCode < 10000 OR tyAlmData.udiCode > 10299 THEN
			tyAlmData.sAlmMsg	:= 'Unknown';
			tyAlmData.sRcyMsg	:= 'Unknown';
		ELSE
			tyAlmData.sAlmMsg	:= a_tyAlmText[tyAlmData.udiCode].sAlmText;
			tyAlmData.sRcyMsg	:= a_tyAlmText[tyAlmData.udiCode].sRcyText;
		END_IF

		sStatTxt	:= tyAlmData.sAlmMsg;

	ELSIF bRstErr AND (tyAlmData.udiCode <> 0) THEN

		tyAlmData.udiCode	:= 0;
		tyAlmData.eSeverity	:= AlmSeverityNA;
		tyAlmData.sAlmMsg	:= '';
		tyAlmData.sRcyMsg	:= '';
		tyAlmData.bAlm		:= FALSE;
		sStatTxt	:= a_sStatText[eStat];

	END_IF

END_ACTION
```

#### Act_Alarm1.st - Do Not Change!!!
```iecst
(** 2020-03-16 **)
ACTION Act_Alarm1:

	//Error
	IF EDGEPOS(eStatus1 = Error) THEN

		tyAlmData1.sProgNm		:= p_sProgNm;
		tyAlmData1.udiCode		:= udiStatus1;
		tyAlmData1.eSeverity	:= AlmSeverityError;
		tyAlmData1.udiRunTime	:= tyAlmData1.udiRunTime + 1;
		tyAlmData1.bAlm			:= TRUE;
		tyAlmData1.udiModuleNum  := udiModuleNum;
		g_sAWOpenProgNm			:= p_sProgNm;

		//Get Error Message
		IF tyAlmData1.udiCode < 10000 OR tyAlmData1.udiCode > 10099 THEN
			tyAlmData1.sAlmMsg	:= 'Unknown';
			tyAlmData1.sRcyMsg	:= 'Unknown';
		ELSE
			tyAlmData1.sAlmMsg	:= a_tyAlmText[tyAlmData1.udiCode].sAlmText;
			tyAlmData1.sRcyMsg	:= a_tyAlmText[tyAlmData1.udiCode].sRcyText;
		END_IF

		sStatTxt	:= tyAlmData1.sAlmMsg;

	ELSIF bRstErr AND (tyAlmData1.udiCode <> 0) THEN

		tyAlmData1.udiCode		:= 0;
		tyAlmData1.eSeverity	:= AlmSeverityNA;
		tyAlmData1.sAlmMsg		:= '';
		tyAlmData1.sRcyMsg		:= '';
		tyAlmData1.bAlm			:= FALSE;
		sStatTxt	:= a_sStatText[eStat];

	END_IF

END_ACTION
```

#### Act_Alarm2.st - Do Not Change!!!
```iecst
(** 2020-03-16 **)
ACTION Act_Alarm2:

	//Error
	IF EDGEPOS(eStatus2 = Error) THEN

		tyAlmData2.sProgNm		:= p_sProgNm;
		tyAlmData2.udiCode		:= udiStatus2;
		tyAlmData2.eSeverity	:= AlmSeverityError;
		tyAlmData2.udiRunTime	:= tyAlmData2.udiRunTime + 1;
		tyAlmData2.bAlm			:= TRUE;
		tyAlmData2.udiModuleNum  := udiModuleNum;
		g_sAWOpenProgNm		:= p_sProgNm;

		//Get Error Message
		IF tyAlmData2.udiCode < 10000 OR tyAlmData2.udiCode > 10099 THEN
			tyAlmData2.sAlmMsg	:= 'Unknown';
			tyAlmData2.sRcyMsg	:= 'Unknown';
		ELSE
			tyAlmData2.sAlmMsg	:= a_tyAlmText[tyAlmData2.udiCode].sAlmText;
			tyAlmData2.sRcyMsg	:= a_tyAlmText[tyAlmData2.udiCode].sRcyText;
		END_IF

		sStatTxt	:= tyAlmData2.sAlmMsg;

	ELSIF bRstErr AND (tyAlmData2.udiCode <> 0) THEN

		tyAlmData2.udiCode		:= 0;
		tyAlmData2.eSeverity	:= AlmSeverityNA;
		tyAlmData2.sAlmMsg		:= '';
		tyAlmData2.sRcyMsg		:= '';
		tyAlmData2.bAlm			:= FALSE;
		sStatTxt	:= a_sStatText[eStat];

	END_IF

END_ACTION
```

#### Act_Alarm3.st - Do Not Change!!!
```iecst
(** 2020-03-16 **)
ACTION Act_Alarm3:

	//Error
	IF EDGEPOS(eStatus3 = Error) THEN

		tyAlmData3.sProgNm		:= p_sProgNm;
		tyAlmData3.udiCode		:= udiStatus3;
		tyAlmData3.eSeverity	:= AlmSeverityError;
		tyAlmData3.udiRunTime	:= tyAlmData3.udiRunTime + 1;
		tyAlmData3.bAlm			:= TRUE;
		tyAlmData3.udiModuleNum := udiModuleNum;
		g_sAWOpenProgNm			:= p_sProgNm;

		//Get Error Message
		IF tyAlmData3.udiCode < 10000 OR tyAlmData3.udiCode > 10099 THEN
			tyAlmData3.sAlmMsg	:= 'Unknown';
			tyAlmData3.sRcyMsg	:= 'Unknown';
		ELSE
			tyAlmData3.sAlmMsg	:= a_tyAlmText[tyAlmData3.udiCode].sAlmText;
			tyAlmData3.sRcyMsg	:= a_tyAlmText[tyAlmData3.udiCode].sRcyText;
		END_IF

		sStatTxt	:= tyAlmData3.sAlmMsg;

	ELSIF bRstErr AND (tyAlmData3.udiCode <> 0) THEN

		tyAlmData3.udiCode		:= 0;
		tyAlmData3.eSeverity	:= AlmSeverityNA;
		tyAlmData3.sAlmMsg		:= '';
		tyAlmData3.sRcyMsg		:= '';
		tyAlmData3.bAlm			:= FALSE;
		sStatTxt	:= a_sStatText[eStat];

	END_IF

END_ACTION
```

#### InputRef.var - Do Not Change!!!
```iecst
(*2020-10-06*)
(**)
(*General*)
VAR
	p_eAct : REFERENCE TO eAWAction;
	p_udiRstErr : REFERENCE TO UDINT;
	p_bPrep : REFERENCE TO BOOL;
	p_bEn : REFERENCE TO BOOL;
	p_bDis : REFERENCE TO BOOL;
END_VAR
(**)
(*Configuration*)
VAR
	p_bOps : REFERENCE TO BOOL;
	p_bManual : REFERENCE TO BOOL;
	p_diWidthAtHmPos : REFERENCE TO DINT;
	p_tyTuning : REFERENCE TO tyMotionCANTuning;
	p_diGoWidth : REFERENCE TO DINT;
	p_diJogVelInUMPS : REFERENCE TO DINT;
	p_diMovePosInUM : REFERENCE TO DINT;
	p_diMoveDistInUM : REFERENCE TO DINT;
	p_diMoveVelInUMPS : REFERENCE TO DINT;
	p_diMoveAcc : REFERENCE TO DINT;
	p_diMoveDec : REFERENCE TO DINT;
	p_diMinAbsPosInUM : REFERENCE TO DINT;
	p_diMaxAbsPosInUM : REFERENCE TO DINT;
	p_diMinWidthInUM : REFERENCE TO DINT;
	p_diMaxWidthInUM : REFERENCE TO DINT;
	p_diWidthOffsetInUM : REFERENCE TO DINT;
	p_bInletSensor : REFERENCE TO BOOL;
	p_bOutletSensor : REFERENCE TO BOOL;
	p_bClearSensor : REFERENCE TO BOOL;
	p_bMiddleSensor : REFERENCE TO BOOL;
	p_bClamp2Sensor : REFERENCE TO BOOL;
	p_bClamp3Sensor : REFERENCE TO BOOL;
	p_bInterruptSensor : REFERENCE TO BOOL;
	p_bOpenInterruptSensor : REFERENCE TO BOOL;
	p_bCloseInterruptSensor : REFERENCE TO BOOL;
	p_bSafetyInterruptSen : REFERENCE TO BOOL;
	p_bDir : REFERENCE TO BOOL;
	p_bDirBl : REFERENCE TO BOOL;
	p_bNoIndexPulse : REFERENCE TO BOOL;
	p_usiNode : REFERENCE TO USINT;
	p_sDevice : REFERENCE TO STRING[3];
	p_sProgNm : REFERENCE TO STRING[15];
	p_diMoveBacklashDistInUM : REFERENCE TO DINT;
	p_diPitchInUM : REFERENCE TO DINT;
	p_tyParamInHm : REFERENCE TO tyMotionCANParamInHm;
	p_tyParamInConvert : REFERENCE TO tyMotionCANParamInConvert;
	p_bNtSettingsLoadDone : REFERENCE TO BOOL;
	p_bOpsAWStepMove : REFERENCE TO BOOL;
	p_eNtParamMotorType : REFERENCE TO eServoMotorType;
	p_bInletShutterCloseRS : REFERENCE TO BOOL;
	p_bOutletShutterCloseRS : REFERENCE TO BOOL;
	p_bInletShutterPrep : REFERENCE TO BOOL;
	p_bInletShutterDis : REFERENCE TO BOOL;
	p_bOutletShutterPrep : REFERENCE TO BOOL;
	p_bOutletShutterDis : REFERENCE TO BOOL;
END_VAR
```

#### Local.var - Do Not Change!!!
```iecst
(*2020-10-06*)
(**)
(*Local Action, State & Status*)
VAR
	eAct : eAWAction := AWActIdle;
	eStat : eAWAction := AWActIdle;
	eMainStatus : eFBStatus := Idle;
	eStatus : eFBStatus := Idle;
	eStatus1 : eFBStatus := Idle;
	eStatus2 : eFBStatus := Idle;
	eStatus3 : eFBStatus := Idle;
	udiStatus : UDINT := 0;
	udiStatus1 : UDINT := 0;
	udiStatus2 : UDINT := 0;
	udiStatus3 : UDINT := 0;
	sStatTxt : STRING[200] := '';
	a_sStatText : ARRAY[0..50] OF STRING[200] := ['Idling','Going Width','Full Homing','Powering On','Powering Off','Homing','Moving Absolute','Moving Relative','Jogging Open','Jogging Close','Jogging Stop','Resetting Axis Error','Stopping','Writing SDO','Background Starting Module OK Check','Background Stopping Module OK Check','Going Width And Power Off','Reset Servo Module Node',33('')];
END_VAR
(**)
(*Local Alarm*)
VAR
	tyAlmData : tyAlmDat;
	tyAlmData1 : tyAlmDat;
	tyAlmData2 : tyAlmDat;
	tyAlmData3 : tyAlmDat;
	a_tyAlmText : ARRAY[10000..10299] OF tyAlmTxt := [(sAlmText:='Axis Move Abnormally By External Force',sRcyText:='Servo Motor Abnormal Operation. Reset And Resume Operation. If The Problem Persists, Please Contact Nutek For A Possible Solution.'),(sAlmText:='CANOpen Communication Error, ModuleOK Not TRUE',sRcyText:='Fail While Read/Write Data. Reset The Error And Resume Operation.'),(sAlmText:='Power On Time Out While Going New Width',sRcyText:='Timeout Expired Before Operation Completed. Reset And Resume Operation.'),(sAlmText:='Homing Time Out While Going New Width',sRcyText:='Timeout Expired Before Operation Completed. Reset And Resume Operation.'),(sAlmText:='Move Absolute Time Out While Going New Width',sRcyText:='Timeout Expired Before Operation Completed. Reset And Resume Operation.'),(sAlmText:='Stop Motion Time Out While Going New Width',sRcyText:='Timeout Expired Before Operation Completed. Reset And Resume Operation.'),(sAlmText:='Axis Error Reset Failed While Going New Width',sRcyText:='Axis Error Reset Failed. Please Retry Again Reset Operation. If The Problem Persists, Please Contact Nutek For A Possible Solution.'),(sAlmText:='Axis Error Occur In Move Absolute While Going New Width',sRcyText:='Servo Motor Abnormal Operation. Reset And Resume Operation. If The Problem Persists, Please Contact Nutek For A Possible Solution.'),(sAlmText:='Axis Error Occur In Homing While Going New Width',sRcyText:='Servo Motor Abnormal Operation. Reset And Resume Operation. If The Problem Persists, Please Contact Nutek For A Possible Solution.'),(sAlmText:='Homing Done But Home Flag Is Not Activated While Going New Width',sRcyText:='Servo Motor Abnormal Operation. Reset And Resume Operation. If The Problem Persists, Please Contact Nutek For A Possible Solution.'),(sAlmText:='Forward Limit Activated In Homing While Going New Width',sRcyText:='Forward Limit Switch Is Activated. Reset The Error By Operate The Motor Backwards.'),(sAlmText:='Reverse Limit Activated In Homing While Going New Width',sRcyText:='Reverse Limit Switch Is Activated. Reset The Error By Operate The Motor Backwards.'),(sAlmText:='Forward Limit Activated In Move Absolute While Going New Width',sRcyText:='Forward Limit Switch Is Activated. Reset The Error By Operate The Motor Backwards.'),(sAlmText:='Reverse Limit Activated In Move Absolute While Going New Width',sRcyText:='Reverse Limit Switch Is Activated. Reset The Error By Operate The Motor Backwards.'),(sAlmText:='Power On Time Out While Full Homing',sRcyText:='Timeout Expired Before Operation Completed. Reset And Resume Operation.'),(sAlmText:='Homing Time Out While Full Homing',sRcyText:='Timeout Expired Before Operation Completed. Reset And Resume Operation.'),(sAlmText:='Stop Motion Time Out While Full Homing',sRcyText:='Timeout Expired Before Operation Completed. Reset And Resume Operation.'),(sAlmText:='Axis Error Reset Failed While Full Homing',sRcyText:='Axis Error Reset Failed. Please Retry Again Reset Operation. If The Problem Persists, Please Contact Nutek For A Possible Solution.'),(sAlmText:='Axis Error Occur In Homing While Full Homing',sRcyText:='Servo Motor Abnormal Operation. Reset And Resume Operation. If The Problem Persists, Please Contact Nutek For A Possible Solution.'),(sAlmText:='Homing Done But Home Flag Is Not Activated While Full Homing',sRcyText:='Servo Motor Abnormal Operation. Reset And Resume Operation. If The Problem Persists, Please Contact Nutek For A Possible Solution.'),(sAlmText:='Forward Limit Activated In Homing While Full Homing',sRcyText:='Forward Limit Switch Is Activated. Reset The Error By Operate The Motor Backwards.'),(sAlmText:='Reverse Limit Activated In Homing While Full Homing',sRcyText:='Reverse Limit Switch Is Activated. Reset The Error By Operate The Motor Backwards.'),(sAlmText:='Power On Time Out',sRcyText:='Timeout Expired Before Operation Completed. Reset And Resume Operation.'),(sAlmText:='Power Off Time Out',sRcyText:='Timeout Expired Before Operation Completed. Reset And Resume Operation.'),(sAlmText:='Homing Time Out',sRcyText:='Timeout Expired Before Operation Completed. Reset And Resume Operation.'),(sAlmText:='Move Absolute Time Out',sRcyText:='Timeout Expired Before Operation Completed. Reset And Resume Operation.'),(sAlmText:='Move Relative Time Out',sRcyText:='Timeout Expired Before Operation Completed. Reset And Resume Operation.'),(sAlmText:='Stop Motion Time Out',sRcyText:='Timeout Expired Before Operation Completed. Reset And Resume Operation.'),(sAlmText:='SDO Write Error',sRcyText:='Fail While Write Data. Reset The Error And Resume Operation.'),(sAlmText:='Request Absolute Position Out Of Range',sRcyText:='Request Absolute Position Does Not Fall Within The Expected Range.'),(sAlmText:='Inlet Sensor Interrupt Auto Width Movement',sRcyText:='Operation Stop Due To The Interruption Of Sensor While Auto Width Moving. Solve The Interruption To Resume Operation.'),(sAlmText:='Outlet Sensor Interrupt Auto Width Movement',sRcyText:='Operation Stop Due To The Interruption Of Sensor While Auto Width Moving. Solve The Interruption To Resume Operation.'),(sAlmText:='Clear Sensor Interrupt Auto Width Movement',sRcyText:='Operation Stop Due To The Interruption Of Sensor While Auto Width Moving. Solve The Interruption To Resume Operation.'),(sAlmText:='Middle Sensor Interrupt Auto Width Movement',sRcyText:='Operation Stop Due To The Interruption Of Sensor While Auto Width Moving. Solve The Interruption To Resume Operation.'),(sAlmText:='Sensor Interrupt Auto Width Movement',sRcyText:='Operation Stop Due To The Interruption Of Sensor While Auto Width Moving. Solve The Interruption To Resume Operation.'),(sAlmText:='Power On Time Out While Going New Width And Off',sRcyText:='Timeout Expired Before Operation Completed. Reset And Resume Operation.'),(sAlmText:='Homing Time Out While Going New Width And Off',sRcyText:='Timeout Expired Before Operation Completed. Reset And Resume Operation.'),(sAlmText:='Move Absolute Time Out While Going New Width And Off',sRcyText:='Timeout Expired Before Operation Completed. Reset And Resume Operation.'),(sAlmText:='Stop Motion Time Out While Going New Width And Off',sRcyText:='Timeout Expired Before Operation Completed. Reset And Resume Operation.'),(sAlmText:='Axis Error Reset Failed While Going New Width And Off',sRcyText:='Axis Error Reset Failed. Please Retry Again Reset Operation. If The Problem Persists, Please Contact Nutek For A Possible Solution.'),(sAlmText:='Axis Error Occur In Move Absolute While Going New Width And Off',sRcyText:='Servo Motor Abnormal Operation. Reset And Resume Operation. If The Problem Persists, Please Contact Nutek For A Possible Solution.'),(sAlmText:='Axis Error Occur In Homing While Going New Width And Off',sRcyText:='Servo Motor Abnormal Operation. Reset And Resume Operation. If The Problem Persists, Please Contact Nutek For A Possible Solution.'),(sAlmText:='Homing Done But Home Flag Is Not Activated While Going New Width And Off',sRcyText:='Servo Motor Abnormal Operation. Reset And Resume Operation. If The Problem Persists, Please Contact Nutek For A Possible Solution.'),(sAlmText:='Forward Limit Activated In Homing While Going New Width And Off',sRcyText:='Forward Limit Switch Is Activated. Reset The Error By Operate The Motor Backwards.'),(sAlmText:='Reverse Limit Activated In Homing While Going New Width And Off',sRcyText:='Reverse Limit Switch Is Activated. Reset The Error By Operate The Motor Backwards.'),(sAlmText:='Forward Limit Activated In Move Absolute While Going New Width And Off',sRcyText:='Forward Limit Switch Is Activated. Reset The Error By Operate The Motor Backwards.'),(sAlmText:='Reverse Limit Activated In Move Absolute While Going New Width And Off',sRcyText:='Reverse Limit Switch Is Activated. Reset The Error By Operate The Motor Backwards.'),2((sAlmText:='Sensor Interrupt Auto Width Movement',sRcyText:='Operation Stop Due To The Interruption Of Sensor While Auto Width Moving. Solve The Interruption To Resume Operation.')),249((0)),(sAlmText:='Forward Limit Activated',sRcyText:='Forward Limit Switch Is Activated. Reset The Error By Operate The Motor Backwards.'),(sAlmText:='Reverse Limit Activated',sRcyText:='Reverse Limit Switch Is Activated. Reset The Error By Operate The Motor Backwards.')];
END_VAR
(**)
(*Local Output*)
VAR
	tyParamOut : tyMotionCANParamOut;
	sAxisErrTxt : STRING[80];
	bWidthPosDiff : BOOL;
	bJogOpen : BOOL;
	bJogClose : BOOL;
	bJogging : BOOL;
	bOpenSen : BOOL;
	bCloseSen : BOOL;
END_VAR
(**)
(*Local Input*)
VAR
	udiRstErr : UDINT := 0;
	bPrep : BOOL := TRUE;
	bEn : BOOL := TRUE;
	bDis : BOOL := FALSE;
	bOps : BOOL := FALSE;
	bManual : BOOL := FALSE;
	diWidthAtHmPos : DINT := 400;
	tyTuning : tyMotionCANTuning;
	diGoWidth : DINT := 150;
	diJogVelInUMPS : DINT := 10000;
	diMovePosInUM : DINT := 0;
	diMoveDistInUM : DINT := 0;
	diMoveVelInUMPS : DINT := 10000;
	diMoveAcc : DINT := 500;
	diMoveDec : DINT := 500;
	diMinAbsPosInUM : DINT := -3000;
	diMaxAbsPosInUM : DINT := 10000000;
	diMinWidthInUM : DINT := 70000;
	diMaxWidthInUM : DINT := 460000;
	diWidthOffsetInUM : DINT := 0;
	bInletSensor : BOOL;
	bOutletSensor : BOOL;
	bClearSensor : BOOL;
	bMiddleSensor : BOOL;
	bClamp2Sensor : BOOL;
	bClamp3Sensor : BOOL;
	bInterruptSensor : BOOL;
	bOpenInterruptSensor : BOOL;
	bCloseInterruptSensor : BOOL;
	bDir : BOOL;
	bDirBl : BOOL;
	bNoIndexPulse : BOOL;
	usiNode : USINT;
	sDevice : STRING[3];
	sProgNm : STRING[15] := 'AWOpen';
	diMoveBacklashDistInUM : DINT := 3000;
	diPitchInUM : DINT := 3000;
	tyParamInHm : tyMotionCANParamInHm;
	tyParamInConvert : tyMotionCANParamInConvert := (diPitchInUM:=3000);
	bNtSettingsLoadDone : BOOL := TRUE;
	eMotorType : eServoMotorType := DeltaAsdaA2;
END_VAR
(**)
(*Local*)
VAR
	bRstErr : BOOL;
	udiRstErrOld : UDINT;
	bInitDone : BOOL;
	bInitialDone : BOOL;
	bModuleOKChk : BOOL := TRUE;
	bModuleOK : BOOL;
	bModuleNotOK : BOOL := TRUE;
	bModuleNotOKLock : BOOL;
	bNotInterruptible : BOOL;
	diActualPosInUMOld : DINT;
	usiRstStep : USINT := 0;
	usiStep : USINT;
	usiCount : USINT;
	fbTm : TON := (PT:=T#2s);
	fbServoModuleNotOk : TON := (IN:=FALSE,PT:=T#2s);
	fbServoModuleOk : TON := (IN:=FALSE,PT:=T#5s);
	fbRstNodeTimer : TON := (PT:=T#3s);
	tyParamInMove : tyMotionCANParamInMove;
	tyParamInDriver : tyMotionCANDriverIn;
	tyParamOutDriver : tyMotionCANDriverOut := (siModOfOpt_6060:=6);
	fbStop : fbMotionCANStop;
	fbRstAxisErr : fbMotionCANRstAxisErr;
	fbJog : fbMotionCANJog;
	fbMovRel : fbMotionCANMovRel;
	fbMovAbs : fbMotionCANMovAbs;
	fbHoming : fbMotionCANHoming;
	fbPwrOff : fbMotionCANPwrOff;
	fbPwrOn : fbMotionCANPwrOn;
	fbFullHm : fbMotionCANFullHm;
	fbFullMovAbs : fbMotionCANFullMovAbs;
	fbFullMovAbsBl : fbMotionCANFullMovAbsBl;
	fbModuleOK : fbMotionCANModuleOK;
	fbSDOWrite : fbCANSDOWriteArrayParam;
	bInletShutterCloseRS : BOOL;
	bOutletShutterCloseRS : BOOL;
	bInletShutterPrep : BOOL;
	bInletShutterDis : BOOL;
	bOutletShutterPrep : BOOL;
	bOutletShutterDis : BOOL;
	udiModuleNum : UDINT := 1;
END_VAR
```

### DInput.var - Change By Project
```iecst
(*2020-10-07*)
(**)
(*Constant*)
VAR CONSTANT
	c_udiDInputMax : UDINT := 40; (*Constant Digital Input Quantity (+1 For Damaged) (+1 For Spare)*)
END_VAR
(**)
(*Action & State & Status*)
(**)
(*Alarm*)
VAR
	p_DIAlmData1 : UDINT;
	p_DIAlmData2 : UDINT;
END_VAR
(**)
(*Output*)
VAR
	p_DI : UDINT;
	p_DISafetyRlySig : UDINT;
	p_DIEStopSig : UDINT;
	p_DICoverSWSig : UDINT;
	p_DIUBA : UDINT;
	p_DIUBAStat : UDINT;
	p_DIDSB : UDINT;
	p_DIUBA2 : UDINT;
	p_DIUBAStat2 : UDINT;
	p_DIConvLftSen : UDINT;
	p_DIConvRgtSen : UDINT;
	p_DIPressureSW : UDINT;
	p_DIThermalPrtSig : UDINT;
	p_DIUSWidthChkSen : UDINT;
	p_DIUSWidthChkSen1 : UDINT;
	p_DIDSWidthChkSen : UDINT;
	p_DIInvertHomeSen : UDINT;
	p_DIInvertRemoteSen : UDINT;
	p_DICoatingSen : UDINT;
	p_DIInShutterOpenRS : UDINT;
	p_DIInShutterCloseRS : UDINT;
	p_DIOutShutterOpenRS : UDINT;
	p_DIOutShutterCloseRS : UDINT;
	p_DIClamp2Sen : UDINT;
	p_DIClamp3Sen : UDINT;
	p_DIClampRS1 : UDINT;
	p_DIUnClampRS1 : UDINT;
	p_DIClampRS2 : UDINT;
	p_DIUnClampRS2 : UDINT;
	p_DIClampRS3 : UDINT;
	p_DIUnClampRS3 : UDINT;
	p_DICoverSWSig2 : UDINT;
	p_DIUnlockCoverSigFromDS : UDINT;
	p_DIUnlockSafetySigFromDS : UDINT;
	p_DIUnlockSafetySigFromUS : UDINT;
	p_DIUnlockCoverSigFromUS : UDINT;
END_VAR
```

### DInput.typ - Change By Project
```iecst
(*2020-10-08*)
(**)
(*Data*)

TYPE
	tyDigitalInput : 	STRUCT
		bSafetyRlySig : BOOL;
		bEStopSig : BOOL;
		bCoverSWSig : BOOL;
		bUBA : BOOL;
		bUBAStat : BOOL;
		bDSB : BOOL;
		bConvLftSen : BOOL;
		bConvRgtSen : BOOL;
		bPressureSW : BOOL;
		bThermalPrtSig : BOOL;
		bCoatingSen : BOOL;
		bUSWidthChkSen : BOOL;
		bDSWidthChkSen : BOOL;
		bInvertHomeSen : BOOL;
		bInvertRemoteSen : BOOL;
		bInShutterOpenRS : BOOL;
		bInShutterCloseRS : BOOL;
		bOutShutterOpenRS : BOOL;
		bOutShutterCloseRS : BOOL;
		bClamp2Sen : BOOL;
		bClamp3Sen : BOOL;
		bClampRS1 : BOOL;
		bUnClampRS1 : BOOL;
		bClampRS2 : BOOL;
		bUnClampRS2 : BOOL;
		bClampRS3 : BOOL;
		bUnClampRS3 : BOOL;
		bUSWidthChkSen1 : BOOL;
		bCoverSWSig2 : BOOL;
		bSafetySigFromUS : BOOL;
		bSafetySigFromDS : BOOL;
		bUnlockCoverSigFromUS : BOOL;
		bUnlockCoverSigFromDS : BOOL;
		bCoverUnlockPB1 : BOOL;
		bUBA2 : BOOL;
		bUBAStat2 : BOOL;
		bSPARE9 : BOOL;
		bSPARE10 : BOOL;
		bSPARE11 : BOOL;
		bSPARE12 : BOOL;
	END_STRUCT;
	tyDigitalInputSettings : 	STRUCT
		diSafetyRlySig : DINT;
		diEStopSig : DINT;
		diCoverSWSig : DINT;
		diUBA : DINT;
		diUBAStat : DINT;
		diDSB : DINT;
		diConvLftSen : DINT;
		diConvRgtSen : DINT;
		diPressureSW : DINT;
		diCoatingSen : DINT;
		diThermalPrtSig : DINT;
		diUSWidthChkSen : DINT;
		diDSWidthChkSen : DINT;
		diInvertHomeSen : DINT;
		diInvertRemoteSen : DINT;
		diInShutterOpenRS : DINT;
		diInShutterCloseRS : DINT;
		diOutShutterOpenRS : DINT;
		diOutShutterCloseRS : DINT;
		diClamp2Sen : DINT;
		diClamp3Sen : DINT;
		diClampRS1 : DINT;
		diUnClampRS1 : DINT;
		diClampRS2 : DINT;
		diUnClampRS2 : DINT;
		diClampRS3 : DINT;
		diUnClampRS3 : DINT;
		diUSWidthChkSen1 : DINT;
		diCoverSWSig2 : DINT;
		diSafetySigFromUS : DINT;
		diSafetySigFromDS : DINT;
		diUnlockCoverSigFromUS : DINT;
		diUnlockCoverSigFromDS : DINT;
		diCoverUnlockPB1 : DINT;
		diUBA2 : DINT;
		diUBAStat2 : DINT;
		diSPARE9 : DINT;
		diSPARE10 : DINT;
		diSPARE11 : DINT;
		diSPARE12 : DINT;
	END_STRUCT;
END_TYPE
```

### Program Logical/DInput/DInput (IEC, version 1.00.0) - 1.00.0 - NtGeneral v5.00.0 (Anson) (2018-11-23)

#### Init.st - Change By Project
```iecst
(** 2020-10-08 **)
PROGRAM _INIT

	(* Always Change If Project Change *)

	//Pass Address To Global Address For External Use
	//Action, State & Status

	//Alarm
	p_DIAlmData1	:= ADR(tyAlmData1);
	p_DIAlmData2	:= ADR(tyAlmData2);

	//Output
	p_DI							:= ADR(tyDInput);
	p_DISafetyRlySig				:= ADR(tyDInput.bSafetyRlySig);
	p_DIEStopSig					:= ADR(tyDInput.bEStopSig);
	p_DICoverSWSig					:= ADR(tyDInput.bCoverSWSig);
	p_DIUBA							:= ADR(tyDInput.bUBA);
	p_DIUBAStat						:= ADR(tyDInput.bUBAStat);
	p_DIDSB							:= ADR(tyDInput.bDSB);
	p_DIUBA2						:= ADR(tyDInput.bUBA2); //ADD_2023-0032B
	p_DIUBAStat2					:= ADR(tyDInput.bUBAStat2); //ADD_2023-0032B
	p_DIConvLftSen					:= ADR(tyDInput.bConvLftSen);
	p_DIConvRgtSen					:= ADR(tyDInput.bConvRgtSen);
	p_DIThermalPrtSig				:= ADR(tyDInput.bThermalPrtSig);
	p_DIUSWidthChkSen				:= ADR(tyDInput.bUSWidthChkSen);
	p_DIDSWidthChkSen				:= ADR(tyDInput.bDSWidthChkSen);
	p_DIInvertHomeSen				:= ADR(tyDInput.bInvertHomeSen);
	p_DIInvertRemoteSen				:= ADR(tyDInput.bInvertRemoteSen);
	p_DICoatingSen					:= ADR(tyDInput.bCoatingSen);
	p_DIPressureSW					:= ADR(tyDInput.bPressureSW);
	p_DIInShutterOpenRS				:= ADR(tyDInput.bInShutterOpenRS);
	p_DIInShutterCloseRS			:= ADR(tyDInput.bInShutterCloseRS);
	p_DIOutShutterOpenRS			:= ADR(tyDInput.bOutShutterOpenRS);
	p_DIOutShutterCloseRS			:= ADR(tyDInput.bOutShutterCloseRS);
	p_DIClamp2Sen					:= ADR(tyDInput.bClamp2Sen);
	p_DIClamp3Sen					:= ADR(tyDInput.bClamp3Sen);
	p_DIClampRS1					:= ADR(tyDInput.bClampRS1);
	p_DIUnClampRS1					:= ADR(tyDInput.bUnClampRS1);
	p_DIClampRS2					:= ADR(tyDInput.bClampRS2);
	p_DIUnClampRS2					:= ADR(tyDInput.bUnClampRS2);
	p_DIClampRS3					:= ADR(tyDInput.bClampRS3);
	p_DIUnClampRS3					:= ADR(tyDInput.bUnClampRS3);
	p_DIUSWidthChkSen1				:= ADR(tyDInput.bUSWidthChkSen1);

	p_DICoverSWSig2					:= ADR(tyDInput.bCoverSWSig2); // ADD
	p_DIUnlockCoverSigFromDS		:= ADR(tyDInput.bUnlockCoverSigFromDS); // ADD
	p_DIUnlockCoverSigFromUS		:= ADR(tyDInput.bUnlockCoverSigFromUS); // ADD
	p_DIUnlockSafetySigFromDS		:= ADR(tyDInput.bSafetySigFromDS);
	p_DIUnlockSafetySigFromUS		:= ADR(tyDInput.bSafetySigFromUS);
	(* Always Change If Project Change *)

END_PROGRAM
```

#### Act_InitGlobal.st - Change By Project
```iecst
(** 2018-12-10 **)
ACTION Act_InitGlobal:

	(* Always Change If Project Change *)

	//Pass Data To Link

	//Pass Data To Internal Use
	p_udiRstErr ACCESS p_RstErrReset;

	p_tyDISettings ACCESS p_NtParamDISettings;

	p_diConvLftSenOnTm ACCESS p_McParamConvLftSenOnTm;
	p_diConvLftSenOffTm ACCESS p_McParamConvLftSenOffTm;
	p_diConvRgtSenOnTm ACCESS p_McParamConvRgtSenOnTm;
	p_diConvRgtSenOffTm ACCESS p_McParamConvRgtSenOffTm;
	p_bRstErrSafetyRlyRst ACCESS p_RstErrSafetyRlyRst;
	p_sProgNm ACCESS p_NtParamDInputProgNm;

	//For BZ startup sound
	p_bLinkStartupRun ACCESS p_StartupRun;
	p_bHermesCmdInitialCompl ACCESS p_HermesCmdInitialCompl;

	(* Always Change If Project Change *)

END_ACTION
```

#### Cyclic.st - Change By Project
```iecst
(** 2019-03-22 **)
PROGRAM _CYCLIC

	IF bInitDone = FALSE THEN
		bInitDone	:= TRUE;

		Act_InitLocal;
		Act_InitGlobal;

	ELSIF bInitialDone = FALSE THEN
		bInitialDone	:= TRUE;

		Act_Initial;

	ELSE
		IF EDGEPOS(p_bHermesCmdInitialCompl) THEN
			Act_InitialCompl;
		END_IF
		Act_RstErr;
		Act_Background;
		Act_Alarm1;
		Act_Alarm2;

	END_IF

END_PROGRAM
```

#### Act_RstErr.st - Do Not Change!!!
```iecst
(** 2018-12-10 **)
ACTION Act_RstErr:

	IF p_udiRstErr <> udiRstErrOld THEN
		bRstErr			:= TRUE;
		udiRstErrOld	:= p_udiRstErr;
	ELSE
		bRstErr			:= FALSE;
	END_IF

END_ACTION
```

#### Act_InitLocal.st - Change By Project
```iecst
(** 2019-03-25 **)
ACTION Act_InitLocal:

	//Input Reference Link To Local Variable
	p_udiMax ACCESS ADR(c_udiDInputMax);
	p_udiRstErr ACCESS ADR(udiRstErr);
	p_tyDISettings ACCESS ADR(tyDISettings);
	p_sProgNm ACCESS ADR(sProgNm);

	p_diConvLftSenOnTm ACCESS ADR(diConvLftSenOnTm);
	p_diConvLftSenOffTm ACCESS ADR(diConvLftSenOffTm);
	p_diConvRgtSenOnTm ACCESS ADR(diConvRgtSenOnTm);
	p_diConvRgtSenOffTm ACCESS ADR(diConvRgtSenOffTm);

	p_bHermesUSCmdFeaturePause ACCESS ADR(bHermesDummyMem);
	p_bHermesDSCmdFeaturePause ACCESS ADR(bHermesDummyMem);
END_ACTION
```

#### Act_Initial.st - Change By Project
```iecst
(** 2018-12-10 **)
ACTION Act_Initial:

	//Initial

END_ACTION
```

#### Act_InitialCompl.st - Change By Project
```iecst
(** 2018-12-10 **)
ACTION Act_InitialCompl:

	//Initial Completed
//	IF p_HermesUSCmdFeaturePause <> 0 THEN
		p_bHermesUSCmdFeaturePause ACCESS p_HermesUSCmdFeaturePause;
//	END_IF
//	IF p_HermesUSCmdPause <> 0  THEN
		p_tyHermesUSCmdPause ACCESS p_HermesUSCmdPause;
//	END_IF
//	IF p_HermesDSCmdFeaturePause <> 0 THEN
		p_bHermesDSCmdFeaturePause ACCESS p_HermesDSCmdFeaturePause;
//	END_IF
//	IF p_HermesDSCmdPause <> 0 THEN
		p_tyHermesDSCmdPause ACCESS p_HermesDSCmdPause;
//	END_IF

END_ACTION
```

#### Act_Background.st - Change By Project
```iecst
(** 2020-10-08 **)
ACTION Act_Background:

	//Digital Input Mapping With Physical Input
	IF p_tyDISettings.diSafetyRlySig > 0 AND p_tyDISettings.diSafetyRlySig <= UDINT_TO_DINT(p_udiMax) THEN
		tyDInput.bSafetyRlySig	:= a_bPhysicalDI[p_tyDISettings.diSafetyRlySig];
	ELSE
		tyDInput.bSafetyRlySig	:= TRUE;
	END_IF

	IF p_tyDISettings.diEStopSig > 0 AND p_tyDISettings.diEStopSig <= UDINT_TO_DINT(p_udiMax) THEN
		tyDInput.bEStopSig	:= a_bPhysicalDI[p_tyDISettings.diEStopSig];
	ELSE
		tyDInput.bEStopSig	:= TRUE;
	END_IF

	IF p_tyDISettings.diCoverSWSig > 0 AND p_tyDISettings.diCoverSWSig <= UDINT_TO_DINT(p_udiMax) THEN
		tyDInput.bCoverSWSig	:= a_bPhysicalDI[p_tyDISettings.diCoverSWSig];
	ELSE
		tyDInput.bCoverSWSig	:= TRUE;
	END_IF

	IF p_tyDISettings.diUBA > 0 AND p_tyDISettings.diUBA <= UDINT_TO_DINT(p_udiMax) THEN
		tyDInput.bUBA	:= a_bPhysicalDI[p_tyDISettings.diUBA];
	ELSE
		tyDInput.bUBA	:= FALSE;
	END_IF

	IF p_tyDISettings.diUBAStat > 0 AND p_tyDISettings.diUBAStat <= UDINT_TO_DINT(p_udiMax) THEN
		tyDInput.bUBAStat	:= a_bPhysicalDI[p_tyDISettings.diUBAStat];
	ELSE
		tyDInput.bUBAStat	:= FALSE;
	END_IF

	IF p_tyDISettings.diDSB > 0 AND p_tyDISettings.diDSB <= UDINT_TO_DINT(p_udiMax) THEN
		tyDInput.bDSB	:= a_bPhysicalDI[p_tyDISettings.diDSB];
	ELSE
		tyDInput.bDSB	:= FALSE;
	END_IF

	IF p_tyDISettings.diUBA2 > 0 AND p_tyDISettings.diUBA2 <= UDINT_TO_DINT(p_udiMax) THEN
		tyDInput.bUBA2	:= a_bPhysicalDI[p_tyDISettings.diUBA2];
	ELSE
		tyDInput.bUBA2	:= FALSE;
	END_IF

	IF p_tyDISettings.diUBAStat2 > 0 AND p_tyDISettings.diUBAStat2 <= UDINT_TO_DINT(p_udiMax) THEN
		tyDInput.bUBAStat2	:= a_bPhysicalDI[p_tyDISettings.diUBAStat2];
	ELSE
		tyDInput.bUBAStat2	:= FALSE;
	END_IF

	IF p_tyDISettings.diConvLftSen > 0 AND p_tyDISettings.diConvLftSen <= UDINT_TO_DINT(p_udiMax) THEN
		//Digital Input Filter
		fbConvLftSigFltr.tSigOnFltrTm	:= DINT_TO_TIME(p_diConvLftSenOnTm);
		fbConvLftSigFltr.tSigOffFltrTm	:= DINT_TO_TIME(p_diConvLftSenOffTm);
		fbConvLftSigFltr(bSigIn := a_bPhysicalDI[p_tyDISettings.diConvLftSen]);
		tyDInput.bConvLftSen	:= fbConvLftSigFltr.bSigOut;
	ELSE
		tyDInput.bConvLftSen	:= FALSE;
	END_IF

	IF p_tyDISettings.diConvRgtSen > 0 AND p_tyDISettings.diConvRgtSen <= UDINT_TO_DINT(p_udiMax) THEN
		//Digital Input Filter
		fbConvRgtSigFltr.tSigOnFltrTm	:= DINT_TO_TIME(p_diConvRgtSenOnTm);
		fbConvRgtSigFltr.tSigOffFltrTm	:= DINT_TO_TIME(p_diConvRgtSenOffTm);
		fbConvRgtSigFltr(bSigIn := a_bPhysicalDI[p_tyDISettings.diConvRgtSen]);
		tyDInput.bConvRgtSen	:= fbConvRgtSigFltr.bSigOut;
	ELSE
		tyDInput.bConvRgtSen	:= FALSE;
	END_IF

	IF p_tyDISettings.diThermalPrtSig > 0 AND p_tyDISettings.diThermalPrtSig <= UDINT_TO_DINT(p_udiMax) THEN
		tyDInput.bThermalPrtSig	:= a_bPhysicalDI[p_tyDISettings.diThermalPrtSig];
	ELSE
		tyDInput.bThermalPrtSig	:= TRUE;
	END_IF

	IF p_tyDISettings.diUSWidthChkSen > 0 AND p_tyDISettings.diUSWidthChkSen <= UDINT_TO_DINT(p_udiMax) THEN
		tyDInput.bUSWidthChkSen	:= a_bPhysicalDI[p_tyDISettings.diUSWidthChkSen];
	ELSE
		tyDInput.bUSWidthChkSen	:= FALSE;
	END_IF

	IF p_tyDISettings.diDSWidthChkSen > 0 AND p_tyDISettings.diDSWidthChkSen <= UDINT_TO_DINT(p_udiMax) THEN
		tyDInput.bDSWidthChkSen	:= a_bPhysicalDI[p_tyDISettings.diDSWidthChkSen];
	ELSE
		tyDInput.bDSWidthChkSen	:= FALSE;
	END_IF

	IF p_tyDISettings.diInvertHomeSen > 0 AND p_tyDISettings.diInvertHomeSen <= UDINT_TO_DINT(p_udiMax) THEN
		tyDInput.bInvertHomeSen	:= a_bPhysicalDI[p_tyDISettings.diInvertHomeSen];
	ELSE
		tyDInput.bInvertHomeSen	:= FALSE;
	END_IF

	IF p_tyDISettings.diInvertRemoteSen > 0 AND p_tyDISettings.diInvertRemoteSen <= UDINT_TO_DINT(p_udiMax) THEN
		tyDInput.bInvertRemoteSen	:= a_bPhysicalDI[p_tyDISettings.diInvertRemoteSen];
	ELSE
		tyDInput.bInvertRemoteSen	:= FALSE;
	END_IF

	IF p_tyDISettings.diCoatingSen > 0 AND p_tyDISettings.diCoatingSen <= UDINT_TO_DINT(p_udiMax) THEN
		tyDInput.bCoatingSen	:= a_bPhysicalDI[p_tyDISettings.diCoatingSen];
	ELSE
		tyDInput.bCoatingSen	:= FALSE;
	END_IF

	IF p_tyDISettings.diInShutterCloseRS > 0 AND p_tyDISettings.diInShutterCloseRS <= UDINT_TO_DINT(p_udiMax) THEN
		tyDInput.bInShutterCloseRS	:= a_bPhysicalDI[p_tyDISettings.diInShutterCloseRS];
	ELSE
		tyDInput.bInShutterCloseRS	:= FALSE;
	END_IF

	IF p_tyDISettings.diInShutterOpenRS > 0 AND p_tyDISettings.diInShutterOpenRS <= UDINT_TO_DINT(p_udiMax) THEN
		tyDInput.bInShutterOpenRS	:= a_bPhysicalDI[p_tyDISettings.diInShutterOpenRS];
	ELSE
		tyDInput.bInShutterOpenRS	:= FALSE;
	END_IF

	IF p_tyDISettings.diOutShutterCloseRS > 0 AND p_tyDISettings.diOutShutterCloseRS <= UDINT_TO_DINT(p_udiMax) THEN
		tyDInput.bOutShutterCloseRS	:= a_bPhysicalDI[p_tyDISettings.diOutShutterCloseRS];
	ELSE
		tyDInput.bOutShutterCloseRS	:= FALSE;
	END_IF

	IF p_tyDISettings.diOutShutterOpenRS > 0 AND p_tyDISettings.diOutShutterOpenRS <= UDINT_TO_DINT(p_udiMax) THEN
		tyDInput.bOutShutterOpenRS	:= a_bPhysicalDI[p_tyDISettings.diOutShutterOpenRS];
	ELSE
		tyDInput.bOutShutterOpenRS	:= FALSE;
	END_IF

	IF p_tyDISettings.diClamp2Sen > 0 AND p_tyDISettings.diClamp2Sen <= UDINT_TO_DINT(p_udiMax) THEN
		tyDInput.bClamp2Sen	:= a_bPhysicalDI[p_tyDISettings.diClamp2Sen];
	ELSE
		tyDInput.bClamp2Sen	:= FALSE;
	END_IF

	IF p_tyDISettings.diClamp3Sen > 0 AND p_tyDISettings.diClamp3Sen <= UDINT_TO_DINT(p_udiMax) THEN
		tyDInput.bClamp3Sen	:= a_bPhysicalDI[p_tyDISettings.diClamp3Sen];
	ELSE
		tyDInput.bClamp3Sen	:= FALSE;
	END_IF

	IF p_tyDISettings.diClampRS1 > 0 AND p_tyDISettings.diClampRS1 <= UDINT_TO_DINT(p_udiMax) THEN
		tyDInput.bClampRS1	:= a_bPhysicalDI[p_tyDISettings.diClampRS1];
	ELSE
		tyDInput.bClampRS1	:= FALSE;
	END_IF

	IF p_tyDISettings.diUnClampRS1 > 0 AND p_tyDISettings.diUnClampRS1 <= UDINT_TO_DINT(p_udiMax) THEN
		tyDInput.bUnClampRS1	:= a_bPhysicalDI[p_tyDISettings.diUnClampRS1];
	ELSE
		tyDInput.bUnClampRS1	:= FALSE;
	END_IF

	IF p_tyDISettings.diClampRS2> 0 AND p_tyDISettings.diClampRS2<= UDINT_TO_DINT(p_udiMax) THEN
		tyDInput.bClampRS2	:= a_bPhysicalDI[p_tyDISettings.diClampRS2];
	ELSE
		tyDInput.bClampRS2	:= FALSE;
	END_IF

	IF p_tyDISettings.diUnClampRS2> 0 AND p_tyDISettings.diUnClampRS2<= UDINT_TO_DINT(p_udiMax) THEN
		tyDInput.bUnClampRS2	:= a_bPhysicalDI[p_tyDISettings.diUnClampRS2];
	ELSE
		tyDInput.bUnClampRS2	:= FALSE;
	END_IF

	IF p_tyDISettings.diClampRS3> 0 AND p_tyDISettings.diClampRS3<= UDINT_TO_DINT(p_udiMax) THEN
		tyDInput.bClampRS3	:= a_bPhysicalDI[p_tyDISettings.diClampRS3];
	ELSE
		tyDInput.bClampRS3	:= FALSE;
	END_IF

	IF p_tyDISettings.diUnClampRS3> 0 AND p_tyDISettings.diUnClampRS3<= UDINT_TO_DINT(p_udiMax) THEN
		tyDInput.bUnClampRS3	:= a_bPhysicalDI[p_tyDISettings.diUnClampRS3];
	ELSE
		tyDInput.bUnClampRS3	:= FALSE;
	END_IF

	IF p_tyDISettings.diPressureSW > 0 AND p_tyDISettings.diPressureSW <= UDINT_TO_DINT(p_udiMax) THEN
		tyDInput.bPressureSW	:= a_bPhysicalDI[p_tyDISettings.diPressureSW];
	ELSE
		tyDInput.bPressureSW	:= FALSE;
	END_IF

	IF p_tyDISettings.diUSWidthChkSen1 > 0 AND p_tyDISettings.diUSWidthChkSen1 <= UDINT_TO_DINT(p_udiMax) THEN
		tyDInput.bUSWidthChkSen1	:= a_bPhysicalDI[p_tyDISettings.diUSWidthChkSen1];
	ELSE
		tyDInput.bUSWidthChkSen1	:= FALSE;
	END_IF

	// ADD
	IF p_tyDISettings.diCoverSWSig2 > 0 AND p_tyDISettings.diCoverSWSig2 <= UDINT_TO_DINT(p_udiMax) THEN
		tyDInput.bCoverSWSig2	:= a_bPhysicalDI[p_tyDISettings.diCoverSWSig2];
	ELSE
		tyDInput.bCoverSWSig2	:= FALSE;
	END_IF

	IF p_bHermesUSCmdFeaturePause THEN
		tyDInput.bSafetySigFromUS	:= p_tyHermesUSCmdPause.bMachineSafetySigFrom;
	ELSIF (p_tyDISettings.diSafetySigFromUS> 0 AND p_tyDISettings.diSafetySigFromUS<= UDINT_TO_DINT(p_udiMax)) THEN
		tyDInput.bSafetySigFromUS	:= a_bPhysicalDI[p_tyDISettings.diSafetySigFromUS];
	ELSE
		tyDInput.bSafetySigFromUS	:= FALSE;
	END_IF

	IF p_bHermesUSCmdFeaturePause THEN
		tyDInput.bUnlockCoverSigFromUS	:= p_tyHermesUSCmdPause.bUnlockCoverSigFrom;
	ELSIF (p_tyDISettings.diUnlockCoverSigFromUS> 0 AND p_tyDISettings.diUnlockCoverSigFromUS<= UDINT_TO_DINT(p_udiMax)) THEN
		tyDInput.bUnlockCoverSigFromUS	:= a_bPhysicalDI[p_tyDISettings.diUnlockCoverSigFromUS];
	ELSE
		tyDInput.bUnlockCoverSigFromUS	:= FALSE;
	END_IF

	IF p_bHermesDSCmdFeaturePause THEN
		tyDInput.bSafetySigFromDS	:= p_tyHermesDSCmdPause.bMachineSafetySigFrom;
	ELSIF (p_tyDISettings.diSafetySigFromDS> 0 AND p_tyDISettings.diSafetySigFromDS<= UDINT_TO_DINT(p_udiMax)) THEN
		tyDInput.bSafetySigFromDS	:= a_bPhysicalDI[p_tyDISettings.diSafetySigFromDS];
	ELSE
		tyDInput.bSafetySigFromDS	:= FALSE;
	END_IF

	IF p_bHermesDSCmdFeaturePause THEN
		tyDInput.bUnlockCoverSigFromDS	:= p_tyHermesDSCmdPause.bUnlockCoverSigFrom;
	ELSIF (p_tyDISettings.diUnlockCoverSigFromDS> 0 AND p_tyDISettings.diUnlockCoverSigFromDS<= UDINT_TO_DINT(p_udiMax))  THEN
		tyDInput.bUnlockCoverSigFromDS	:= a_bPhysicalDI[p_tyDISettings.diUnlockCoverSigFromDS];
	ELSE
		tyDInput.bUnlockCoverSigFromDS	:= FALSE;
	END_IF

	IF p_tyDISettings.diCoverUnlockPB1> 0 AND p_tyDISettings.diCoverUnlockPB1<= UDINT_TO_DINT(p_udiMax) THEN
		tyDInput.bCoverUnlockPB1	:= a_bPhysicalDI[p_tyDISettings.diCoverUnlockPB1];
	ELSE
		tyDInput.bCoverUnlockPB1	:= FALSE;
	END_IF

	//For Simulation Only
	IF DiagCpuIsSimulated() = TRUE THEN
		tyDInput.bSafetyRlySig	:= TRUE;
		tyDInput.bEStopSig		:= TRUE;
		tyDInput.bCoverSWSig	:= TRUE;
		tyDInput.bThermalPrtSig	:= TRUE;
		tyDInput.bPressureSW	:= TRUE;
	END_IF
	//Estop
	IF (tyDInput.bEStopSig = FALSE) AND (eStatus1 <> Error) THEN
		eStatus1	:= Error;
		udiStatus1	:= 10000;	//Emergency Stop Button Pressed
	END_IF

	//Cover Switch
	IF (tyDInput.bCoverSWSig = FALSE) AND (eStatus2 <> Error) THEN
		eStatus2	:= Error;
		udiStatus2	:= 10001;	//Door / Conver Opened
	END_IF

	IF p_bLinkStartupRun THEN
		fbSafetyRlyRstTm(IN := NOT(p_bRstErrSafetyRlyRst));
		IF (tyDInput.bSafetyRlySig = FALSE) AND fbSafetyRlyRstTm.Q THEN
			bSafetySigErrNoBuz	:= TRUE;
		END_IF
	ELSIF bSafetySigErrNoBuz = FALSE THEN
		fbSafetyRlyRstTm(IN := NOT(p_bRstErrSafetyRlyRst));
		IF (tyDInput.bSafetyRlySig = FALSE) AND (eStatus2<>Error AND eStatus1<>Error) AND fbSafetyRlyRstTm.Q AND tyDInput.bEStopSig AND tyDInput.bCoverSWSig THEN
			eStatus2	:= Error;
			udiStatus2	:= 10002; //Safety Relay Signal is Off
		END_IF
	END_IF

	//Reset Error
	IF (eStatus1 = Error) AND bRstErr THEN
		eStatus1	:= Idle;
		udiStatus1	:= 0;
	END_IF

	IF (eStatus2 = Error) AND bRstErr THEN
		eStatus2	:= Idle;
		udiStatus2	:= 0;
	END_IF

	IF bRstErr AND bSafetySigErrNoBuz THEN
		bSafetySigErrNoBuz	:= FALSE;
	END_IF

//	fbSafetyRlyRstTm (IN := NOT(p_bRstErrSafetyRlyRst));
//	IF (tyDInput.bSafetyRlySig = FALSE) AND (eStatus2 <> Error) AND fbSafetyRlyRstTm.Q AND tyDInput.bEStopSig AND tyDInput.bCoverSWSig THEN
//		eStatus2 := Error;
//		udiStatus2 := 10002;
//	END_IF

END_ACTION
```

#### Act_Alarm1.st - Change By Project
```iecst
(** 2019-03-25 **)
ACTION Act_Alarm1:

	//Error
	IF EDGEPOS(eStatus1 = Error) THEN

		tyAlmData1.sProgNm		:= p_sProgNm;
		tyAlmData1.udiCode		:= udiStatus1;
		tyAlmData1.eSeverity	:= AlmSeverityError;
		tyAlmData1.udiRunTime	:= tyAlmData1.udiRunTime + 1;
		tyAlmData1.bAlm			:= TRUE;
		tyAlmData1.udiModuleNum := udiModuleNum;
		g_sDInputProgNm			:= p_sProgNm;

		//Get Error Message
		IF tyAlmData1.udiCode < 10000 OR tyAlmData1.udiCode > 10099 THEN
			tyAlmData1.sAlmMsg	:= 'Unknown';
			tyAlmData1.sRcyMsg	:= 'Unknown';
		ELSE
			tyAlmData1.sAlmMsg	:= a_tyAlmText[tyAlmData1.udiCode].sAlmText;
			tyAlmData1.sRcyMsg	:= a_tyAlmText[tyAlmData1.udiCode].sRcyText;
		END_IF

	ELSIF bRstErr AND (tyAlmData1.udiCode <> 0) THEN

		tyAlmData1.udiCode		:= 0;
		tyAlmData1.eSeverity	:= AlmSeverityNA;
		tyAlmData1.sAlmMsg		:= '';
		tyAlmData1.sRcyMsg		:= '';
		tyAlmData1.bAlm			:= FALSE;
	END_IF

END_ACTION
```

#### Act_Alarm2.st - Change By Project
```iecst
(** 2019-03-25 **)
ACTION Act_Alarm2:

	//Error
	IF EDGEPOS(eStatus2 = Error) THEN

		tyAlmData2.sProgNm		:= p_sProgNm;
		tyAlmData2.udiCode		:= udiStatus2;
		tyAlmData2.eSeverity	:= AlmSeverityError;
		tyAlmData2.udiRunTime	:= tyAlmData2.udiRunTime + 1;
		tyAlmData2.bAlm			:= TRUE;
		tyAlmData2.udiModuleNum := udiModuleNum;
		g_sDInputProgNm			:= p_sProgNm;

		//Get Error Message
		IF tyAlmData2.udiCode < 10000 OR tyAlmData2.udiCode > 10099 THEN
			tyAlmData2.sAlmMsg	:= 'Unknown';
			tyAlmData2.sRcyMsg	:= 'Unknown';
		ELSE
			tyAlmData2.sAlmMsg	:= a_tyAlmText[tyAlmData2.udiCode].sAlmText;
			tyAlmData2.sRcyMsg	:= a_tyAlmText[tyAlmData2.udiCode].sRcyText;
		END_IF

	ELSIF bRstErr AND (tyAlmData2.udiCode <> 0) THEN

		tyAlmData2.udiCode		:= 0;
		tyAlmData2.eSeverity	:= AlmSeverityNA;
		tyAlmData2.sAlmMsg		:= '';
		tyAlmData2.sRcyMsg		:= '';
		tyAlmData2.bAlm			:= FALSE;
	END_IF

END_ACTION
```

#### InputRef.var - Change By Project
```iecst
(*2019-03-22*)
(**)
(*General*)
VAR
	p_udiMax : REFERENCE TO UDINT;
	p_udiRstErr : REFERENCE TO UDINT;
END_VAR
(**)
(*Configuration*)
VAR
	p_tyDISettings : REFERENCE TO tyDigitalInputSettings;
END_VAR
(**)
VAR
	p_diConvLftSenOnTm : REFERENCE TO DINT;
	p_diConvLftSenOffTm : REFERENCE TO DINT;
	p_diConvRgtSenOnTm : REFERENCE TO DINT;
	p_diConvRgtSenOffTm : REFERENCE TO DINT;
	p_sProgNm : REFERENCE TO STRING[15];
	p_bRstErrSafetyRlyRst : REFERENCE TO BOOL;
END_VAR
(**)
VAR
	p_bLinkStartupRun : REFERENCE TO BOOL;
END_VAR
(* *)
VAR
	p_bHermesCmdInitialCompl : REFERENCE TO BOOL;
	p_bHermesUSCmdFeaturePause : REFERENCE TO BOOL;
	p_tyHermesUSCmdPause : REFERENCE TO tyHermesCommandPause;
	p_bHermesDSCmdFeaturePause : REFERENCE TO BOOL;
	p_tyHermesDSCmdPause : REFERENCE TO tyHermesCommandPause;
END_VAR
```

#### Local.var - Change By Project
```iecst
(*2019-03-25*)
(**)
(*Local Action, State & Status*)
VAR
	eStatus1 : eFBStatus := Idle;
	eStatus2 : eFBStatus := Idle;
	udiStatus1 : UDINT := 0;
	udiStatus2 : UDINT := 0;
END_VAR
(**)
(*Local Alarm*)
VAR
	tyAlmData1 : tyAlmDat;
	tyAlmData2 : tyAlmDat;
	a_tyAlmText : ARRAY[10000..10099] OF tyAlmTxt := [(sAlmText:='Emergency Stop Button Pressed',sRcyText:='Release The Emergency Stop Button And Reset The Error To Resume Operation.'),(sAlmText:='Door / Cover Opened',sRcyText:='Close The Door / Cover Tightly And Resume Operation.'),(sAlmText:='Safety Relay Signal is off',sRcyText:='Reset the Safety Relay'),97(0)];
END_VAR
(**)
(*Local Output*)
VAR
	tyDInput : tyDigitalInput;
END_VAR
(**)
(*Local Input*)
VAR
	udiRstErr : UDINT := 0;
	tyDISettings : tyDigitalInputSettings := (0);
END_VAR
(**)
VAR
	diConvLftSenOnTm : DINT := 50;
	diConvLftSenOffTm : DINT := 50;
	diConvRgtSenOnTm : DINT := 50;
	diConvRgtSenOffTm : DINT := 50;
	sProgNm : STRING[15] := 'DInput';
END_VAR
(**)
(*Local*)
VAR
	bRstErr : BOOL;
	udiRstErrOld : UDINT;
	bInitDone : BOOL;
	bInitialDone : BOOL;
	a_bPhysicalDI : ARRAY[1..c_udiDInputMax] OF BOOL;
	fbConvLftSigFltr : fbSenFltr;
	fbConvRgtSigFltr : fbSenFltr;
	fbSafetyRlyRstTm : TON := (PT:=T#1s);
	udiModuleNum : UDINT := 5751;
	bSafetySigErrNoBuz : BOOL;
	bHermesDummyMem : BOOL;
END_VAR
```

### DOutput.var - Change By Project
```iecst
(*2019-01-08*)
(**)
(*Constant*)
VAR CONSTANT
	c_udiDOutputMax : UDINT := 40; (*Constant Digital Output Quantity (+1 For Damaged)(+1 For Spare)*)
END_VAR
(**)
(*Action & State & Status*)
VAR
	p_DOAct : UDINT;
	p_DOStat : UDINT;
	p_DOStatus : UDINT;
	p_DOStatTxt : UDINT;
END_VAR
(**)
(*Alarm*)
(**)
(*Output*)
VAR
	p_DO : UDINT;
END_VAR
```

### DOutput.typ - Change By Project
```iecst
(*2020-10-08*)
(**)
(*Action*)

TYPE
	eDOAction :
		(
		DOActIdle,
		DOActRstAll,
		DOActSetBypassCoverSwitch,
		DOActRstBypassCoverSwitch
		);
END_TYPE

(**)
(*Data*)

TYPE
	tyDigitalOutput : 	STRUCT
		bSafetyRlyRst : BOOL;
		bTLRed : BOOL;
		bTLAmber : BOOL;
		bTLGreen : BOOL;
		bTLBlue : BOOL;
		bTLWhite : BOOL;
		bBuz : BOOL;
		bCoatingStprRet : BOOL;
		bUSB : BOOL;
		bDBA : BOOL;
		bDBAStat : BOOL;
		bConvMtrCW : BOOL;
		bConvMtrCCW : BOOL;
		bStprUnblkCtrl : BOOL;
		bStprBlkCtrl : BOOL;
		bInvertHome : BOOL;
		bInvertRemote : BOOL;
		bInvertBrake : BOOL;
		bMtrPwrRly : BOOL;
		bClampControl : BOOL;
		bUnclampControl : BOOL;
		bInShutterOpenCtrl : BOOL;
		bInShutterCloseCtrl : BOOL;
		bOutShutterOpenCtrl : BOOL;
		bOutShutterCloseCtrl : BOOL;
		bClamp1Ctrl : BOOL;
		bUnClamp1Ctrl : BOOL;
		bClamp2Ctrl : BOOL;
		bUnClamp2Ctrl : BOOL;
		bClamp3Ctrl : BOOL;
		bUnClamp3Ctrl : BOOL;
		bTopCvrUnlckToDS : BOOL;
		bTopCvrUnlckToUS : BOOL;
		bMachineSafetySigToDS : BOOL;
		bMachineSafetySigToUS : BOOL;
		bCoverPBLED1 : BOOL;
		bBypassTopCover1 : BOOL;
		bSafetyTopCoverSWCoil1 : BOOL;
		bUSB2 : BOOL;
		bSPARE9 : BOOL;
		bSPARE10 : BOOL;
		bSPARE11 : BOOL;
		bSPARE12 : BOOL;
	END_STRUCT;
	tyDigitalOutputSettings : 	STRUCT
		diSafetyRlyRst : DINT;
		diTLRed : DINT;
		diTLAmber : DINT;
		diTLGreen : DINT;
		diTLBlue : DINT;
		diTLWhite : DINT;
		diBuz : DINT;
		diCoatingStprRet : DINT;
		diUSB : DINT;
		diDBA : DINT;
		diDBAStat : DINT;
		diConvMtrCW : DINT;
		diConvMtrCCW : DINT;
		diStprUnblkCtrl : DINT;
		diStprBlkCtrl : DINT;
		diInvertHome : DINT;
		diInvertRemote : DINT;
		diInvertBrake : DINT;
		diMtrPwrRly : DINT;
		diClampControl : DINT;
		diUnclampControl : DINT;
		diInShutterOpenCtrl : DINT;
		diInShutterCloseCtrl : DINT;
		diOutShutterOpenCtrl : DINT;
		diOutShutterCloseCtrl : DINT;
		diClamp1Ctrl : DINT;
		diUnClamp1Ctrl : DINT;
		diClamp2Ctrl : DINT;
		diUnClamp2Ctrl : DINT;
		diClamp3Ctrl : DINT;
		diUnClamp3Ctrl : DINT;
		diTopCvrUnlckToDS : DINT;
		diTopCvrUnlckToUS : DINT;
		diMachineSafetySigToDS : DINT;
		diMachineSafetySigToUS : DINT;
		diCoverPBLED1 : DINT;
		diBypassTopCover1 : DINT;
		diSafetyTopCoverSWCoil1 : DINT;
		diUSB2 : DINT;
		diSPARE9 : DINT;
		diSPARE10 : DINT;
		diSPARE11 : DINT;
		diSPARE12 : DINT;
	END_STRUCT;
END_TYPE
```

### Program Logical/DOutput/DOutput (IEC, version 1.00.0) - 1.00.0 - (Anson) (2018-11-23)

#### Init.st - Change By Project
```iecst
(** 202019-03-25 **)
PROGRAM _INIT

	(* Always Change If Project Change *)

	//Pass Address To Global Address For External Use
	//Action, State & Status
	p_DOStat	:= ADR(eStat);
	p_DOStatus	:= ADR(eStatus);
	p_DOStatTxt	:= ADR(sStatTxt);

	//Alarm

	//Output
	p_DO	:= ADR(tyDOutput);

	(* Always Change If Project Change *)

END_PROGRAM
```

#### Act_InitGlobal.st - Change By Project
```iecst
(** 2020-10-08 **)
ACTION Act_InitGlobal:

	(* Always Change If Project Change *)

	//Pass Data To Link
	p_eLinkOpsInvertInvertCurrPos ACCESS p_OpsInvertInvertCurrPos;
	p_bLinkConvMtrSigOnOrLToR ACCESS p_ConvMtrSigOnOrLToR;
	p_bLinkConvMtrDirOrRToL ACCESS p_ConvMtrDirOrRToL;

	p_bLinkUIConvDCCtrl ACCESS p_UIConvDCCtrl;
//	p_bLinkUIInvertDCCtrl ACCESS p_UIInvertDCCtrl;
	p_usiLinkProdRcpCurrRcpMcMod ACCESS p_ProdRcpCurrRcp1McMod;
	p_eConvStatus ACCESS p_ConvStatus;

	p_bLinkOpsInvertStepInitTwdStpr ACCESS p_OpsInvertStepInitTwdStpr;
	p_bLinkOpsInvertStepInitAwayStpr ACCESS p_OpsInvertStepInitAwayStpr;

	//Pass Data To Internal Use
	p_eAct ACCESS p_UIDOAct;
	p_tyDOSettings ACCESS p_NtParamDOSettings;

	p_bManual ACCESS p_UIUIMnlMod;
	p_bSafetyRlyRst ACCESS p_RstErrSafetyRlyRst;
	p_bTLWhite ACCESS p_TLBuzWhite;
	p_bTLAmber ACCESS p_TLBuzAmber;
	p_bTLGreen ACCESS p_TLBuzGreen;
	p_bTLRed ACCESS p_TLBuzRed;
	p_bTLBlue ACCESS p_TLBuzBlue;
	p_bBuz ACCESS p_TLBuzBeep;
	p_bUSB ACCESS p_USSMEMAUSB;
	p_bDBA ACCESS p_DSSMEMADBA;
	p_bUSB2 ACCESS p_USSMEMA2USB;
	p_bDBAStat ACCESS p_DSSMEMADBAStat;
	p_bStprUnblkCtrl ACCESS p_PneuNoSenStopperRetCtrl;
	p_bStprBlkCtrl ACCESS p_PneuNoSenStopperExtCtrl;
	p_bInvertHome ACCESS p_MotorBrkMtrSigOnOrCW;
	p_bInvertRemote ACCESS p_MotorBrkMtrDirOrCCW;
	p_bInvertBrake ACCESS p_MotorBrkMtrBrkRls;
	p_bClampControl ACCESS p_PneuNoSenClampExtCtrl;
	p_bUnclampControl ACCESS p_PneuNoSenClampRetCtrl;
	p_bInShutterOpenCtrl ACCESS p_Pneu2SenInShutterRetCtrl;
	p_bInShutterCloseCtrl ACCESS p_Pneu2SenInShutterExtCtrl;
	p_bOutShutterOpenCtrl ACCESS p_Pneu2SenOutShutterRetCtrl;
	p_bOutShutterCloseCtrl ACCESS p_Pneu2SenOutShutterExtCtrl;

	//Clamp
	p_bClamp1Ctrl ACCESS p_Pneu2SenClamp1ExtCtrl;
	p_bUnClamp1Ctrl ACCESS p_Pneu2SenClamp1RetCtrl;
	p_bClamp2Ctrl ACCESS p_Pneu2SenClamp2ExtCtrl;
	p_bUnClamp2Ctrl ACCESS p_Pneu2SenClamp2RetCtrl;
	p_bClamp3Ctrl ACCESS p_Pneu2SenClamp3ExtCtrl;
	p_bUnClamp3Ctrl ACCESS p_Pneu2SenClamp3RetCtrl;

	p_tyDI ACCESS p_DI;
	p_bHermesCmdInitialCompl ACCESS p_HermesCmdInitialCompl;

	(* Always Change If Project Change *)

END_ACTION
```

#### Act_LinkAction.st - Change By Project
```iecst
(** 2019-03-29 **)
ACTION Act_LinkAction:

	IF EDGENEG(p_bManual) THEN
		p_eAct	:= DOActIdle;
	END_IF

END_ACTION
```

#### Act_Link.st - Change By Project
```iecst
(** 2019-03-29 **)
ACTION Act_Link:

//	IF p_bLinkUIInvertDCCtrl THEN
//		p_bInvertBrake ACCESS p_UIInvertDCModBrakePress;
//	ELSE
//		p_bInvertBrake ACCESS p_MotorBrkMtrBrkRls;
//	END_IF
	IF p_bManual THEN
		p_bBypsCoverSW1 ACCESS p_UIMnlModBypassTopCover1;			// ADD
		p_bTopCvrUnlckToDS ACCESS p_UIMnlModTopCvrUnlckToDS;			//
		p_bTopCvrUnlckToUS ACCESS p_UIMnlModTopCvrUnlckToUS;			//
		p_bMachineSafetySigToDS ACCESS p_UIMnlModMachineSafetySigToDS;	// ADD
		p_bMachineSafetySigToUS ACCESS p_UIMnlModMachineSafetySigToUS;	// ADD
		p_bSafetyTopCoverSWCoil1 ACCESS p_UIMnlModSafetyTopCoverSWCoil1;	//
		p_bCoverPBLED1 ACCESS p_UIMnlModCoverPBLED1;				//
	ELSE
		p_bBypsCoverSW1 ACCESS p_UIBypassTopCover1 ;			// ADD
		p_bMachineSafetySigToDS ACCESS p_UIMachineSafetySigToDS ;			//
		p_bMachineSafetySigToUS ACCESS  p_UIMachineSafetySigToUS ;			//
		p_bTopCvrUnlckToDS ACCESS p_UITopCvrUnlckToDS;	// ADD
		p_bTopCvrUnlckToUS ACCESS p_UITopCvrUnlckToUS ;	// ADD
		p_bSafetyTopCoverSWCoil1 ACCESS p_UISafetyTopCoverSWCoil1;	//
		p_bCoverPBLED1 ACCESS p_UICoverPBLED1;				//
	END_IF

	IF p_eLinkOpsInvertInvertCurrPos = InvertCurrPosAtRemote THEN

		IF p_eConvStatus = Busy THEN
			p_bConvMtrCW	:= p_bLinkConvMtrDirOrRToL;
			p_bConvMtrCCW  := p_bLinkConvMtrSigOnOrLToR;
		ELSE
			IF p_bManual = TRUE AND p_bLinkUIConvDCCtrl = TRUE THEN
				p_bConvMtrCW	:= p_bLinkConvMtrSigOnOrLToR;
				p_bConvMtrCCW	:= p_bLinkConvMtrDirOrRToL;
			ELSE
				p_bConvMtrCW	:= FALSE;
				p_bConvMtrCCW	:= FALSE;
			END_IF

		END_IF

	ELSIF p_eLinkOpsInvertInvertCurrPos = InvertCurrPosAtHome THEN

		IF p_eConvStatus = Busy THEN
			p_bConvMtrCW	:= p_bLinkConvMtrSigOnOrLToR;
			p_bConvMtrCCW	:= p_bLinkConvMtrDirOrRToL;
		ELSE
			IF p_bManual = TRUE AND p_bLinkUIConvDCCtrl = TRUE THEN
				p_bConvMtrCW	:= p_bLinkConvMtrSigOnOrLToR;
				p_bConvMtrCCW	:= p_bLinkConvMtrDirOrRToL;
			ELSE
				p_bConvMtrCW	:= FALSE;
				p_bConvMtrCCW	:= FALSE;
			END_IF

		END_IF

	ELSE
		p_bConvMtrCW	:= p_bLinkConvMtrSigOnOrLToR;
		p_bConvMtrCCW	:= p_bLinkConvMtrDirOrRToL;
	END_IF

	//Output Invert Bypass/Invert Signal
//	p_bInvertBypsMod	:= p_usiLinkProdRcpCurrRcpMcMod = 0;
//	p_bInvertInvertMod	:= p_usiLinkProdRcpCurrRcpMcMod = 1;

	IF p_tyDI.bSafetyRlySig AND p_tyDI.bCoverSWSig AND p_tyDI.bEStopSig AND p_tyDI.bThermalPrtSig THEN
		p_bMtrPwrRly := TRUE ;
	ELSE
		p_bMtrPwrRly := FALSE;
	END_IF

END_ACTION
```

#### Cyclic.st - Change By Project
```iecst
(** 2019-03-29 **)
PROGRAM _CYCLIC

	IF bInitDone = FALSE THEN
		bInitDone	:= TRUE;

		Act_InitLocal;
		Act_InitGlobal;

	ELSIF bInitialDone = FALSE THEN
		bInitialDone	:= TRUE;

		Act_Initial;

	ELSE
		IF EDGEPOS(p_bHermesCmdInitialCompl) THEN
			Act_InitialCompl;
		END_IF
		Act_LinkAction;
		Act_Action;
		Act_Link;
		Act_Main;
		Act_Background;

	END_IF

END_PROGRAM
```

#### Act_InitLocal.st - Change By Project
```iecst
(** 2020-10-08 **)
ACTION Act_InitLocal:

	//Input Reference Link To Local Variable
	p_udiMax ACCESS ADR(c_udiDOutputMax);
	p_eAct ACCESS ADR(eAct);
	p_tyDOSettings ACCESS ADR(tyDOSettings);
	p_bManual ACCESS ADR(bManual);
	p_bSafetyRlyRst ACCESS ADR(bSafetyRlyRst);
	p_bTLRed ACCESS ADR(bTLRed);
	p_bTLAmber ACCESS ADR(bTLAmber);
	p_bTLGreen ACCESS ADR(bTLGreen);
	p_bTLWhite ACCESS ADR(bTLWhite);
	p_bTLBlue ACCESS ADR(bTLBlue);
	p_bBuz ACCESS ADR(bBuz);
	p_bUSB ACCESS ADR(bUSB);
	p_bDBA ACCESS ADR(bDBA);
	p_bDBAStat ACCESS ADR(bDBAStat);
	p_bUSB2 ACCESS ADR(bUSB2);
	p_bConvMtrCW ACCESS ADR(bConvMtrCW);
	p_bConvMtrCCW ACCESS ADR(bConvMtrCCW);
	p_bStprUnblkCtrl ACCESS ADR(bStprUnblkCtrl);
	p_bStprBlkCtrl ACCESS ADR(bStprBlkCtrl);
	p_bInvertHome ACCESS ADR(bInvertHome);
	p_bInvertRemote ACCESS ADR(bInvertRemote);
	p_bInvertBrake ACCESS ADR(bInvertBrake);
	p_bClampControl ACCESS ADR(bClampControl);
	p_bUnclampControl ACCESS ADR(bUnclampControl);
	p_bMtrPwrRly ACCESS ADR (bMtrPwrRly);
	p_bInShutterOpenCtrl ACCESS ADR(bInShutterOpenCtrl);
	p_bInShutterCloseCtrl ACCESS ADR(bInShutterCloseCtrl);
	p_bOutShutterOpenCtrl ACCESS ADR(bOutShutterOpenCtrl);
	p_bOutShutterCloseCtrl ACCESS ADR(bOutShutterCloseCtrl);
	p_bClamp1Ctrl ACCESS ADR(bClamp1Ctrl);
	p_bUnClamp1Ctrl ACCESS ADR(bUnClamp1Ctrl);
	p_bClamp2Ctrl ACCESS ADR(bClamp2Ctrl);
	p_bUnClamp2Ctrl ACCESS ADR(bUnClamp2Ctrl);
	p_bClamp3Ctrl ACCESS ADR(bClamp3Ctrl);
	p_bUnClamp3Ctrl ACCESS ADR(bUnClamp3Ctrl);

	p_bBypsCoverSW1 ACCESS ADR(bBypassTopCover1);			// ADD
	p_bTopCvrUnlckToDS ACCESS ADR(bTopCvrUnlckToDS);			//
	p_bTopCvrUnlckToUS ACCESS ADR(bTopCvrUnlckToUS);			//
	p_bMachineSafetySigToDS ACCESS ADR(bMachineSafetySigToDS);	// ADD
	p_bMachineSafetySigToUS ACCESS ADR(bMachineSafetySigToUS);	// ADD
	p_bSafetyTopCoverSWCoil1 ACCESS ADR(bSafetyTopCoverSWCoil1);	//
	p_bCoverPBLED1 ACCESS ADR(bCoverPBLED1);				//

	p_bHermesUSCmdFeaturePause ACCESS ADR(bHermesDummyMem);
	p_bHermesDSCmdFeaturePause ACCESS ADR(bHermesDummyMem);
END_ACTION
```

#### Act_InitialCompl.st - Change By Project
```iecst
(** 2018-12-10 **)
ACTION Act_InitialCompl:

	//Initial Completed
//	IF p_HermesUSCmdFeaturePause <> 0 THEN
		p_bHermesUSCmdFeaturePause ACCESS p_HermesUSCmdFeaturePause;
//	END_IF
//	IF p_HermesUSCmdPause <> 0  THEN
		p_tyHermesUSCmdPause ACCESS p_HermesUSCmdPause;
//	END_IF
//	IF p_HermesDSCmdFeaturePause <> 0 THEN
		p_bHermesDSCmdFeaturePause ACCESS p_HermesDSCmdFeaturePause;
//	END_IF
//	IF p_HermesDSCmdPause <> 0 THEN
		p_tyHermesDSCmdPause ACCESS p_HermesDSCmdPause;
//	END_IF
END_ACTION
```

#### Act_Action.st - Do Not Change!!!
```iecst
(** 2019-03-25 **)
ACTION Act_Action:

	//Set p_eAct
	IF eStatus = Idle OR eStatus = Busy OR eStatus = Done THEN
		eStat	:= p_eAct;
	END_IF

END_ACTION
```

#### Act_Main.st - Change By Project
```iecst
(** 2019-01-10 **)
ACTION Act_Main:

	IF eStatOld <> eStat THEN
		sStatTxt	:= a_sStatText[eStat];

		eStatOld	:= eStat;

		eStatus		:= Busy;
	END_IF

	//Main
	CASE eStat OF

		DOActIdle:
			eStatus	:= Idle;

		DOActRstAll:
			IF eStatus = Idle OR eStatus = Busy THEN

//				p_bBypassCoverSwitch	:= FALSE;
				eStatus					:= Done;

			END_IF

		DOActSetBypassCoverSwitch:
			IF eStatus = Idle OR eStatus = Busy THEN

//				p_bBypassCoverSwitch	:= TRUE;
				eStatus					:= Done;

			END_IF

		DOActRstBypassCoverSwitch:
			IF eStatus = Idle OR eStatus = Busy THEN

//				p_bBypassCoverSwitch	:= FALSE;
				eStatus					:= Done;

			END_IF

	END_CASE

END_ACTION
```
